// TwinCAT 3 PLC project LWLine
// Title: LINE_LJ
// Company: Aircom Automotive
// ProjectVersion: 1.0
// ProgramVersion: 3.1.4020.4
// CompilerDefines: VISU_USEWSTRING
// libraries:
//   AirLib_Mach, * (AirCom)
//   AirLib_PIM, * (AirCom)
//   VisuElemBase, * (System)
//   VisuElemMeter, * (System)
//   VisuElems, * (System)
//   VisuElemsSpecialControls, * (System)
//   VisuElemsWinControls, * (System)
//   VisuElemTextEditor, * (System)
//   VisuInputs, * (System)
//   VisuNativeControl, * (System)
//   Tc2_Math, * (Beckhoff Automation GmbH)
//   Tc2_MC2, * (Beckhoff Automation GmbH)
//   Tc2_MC2_Drive, * (Beckhoff Automation GmbH)
//   Tc2_ModbusSrv, * (Beckhoff Automation GmbH)
//   Tc2_SerialCom, * (Beckhoff Automation GmbH)
//   Tc2_TcpIp, * (Beckhoff Automation GmbH)
//   Tc3_Database, * (Beckhoff Automation GmbH)
//   TC3_EL6910_Backup_Restore, * (Beckhoff Automation GmbH)
//   Tc3_EventLogger, * (Beckhoff Automation GmbH)
//   Tc3_Interfaces, * (Beckhoff Automation GmbH)
//   Tc3_Module, * (Beckhoff Automation GmbH)
//   Util, * (System)
//   VisuDialogs, * (System)
//   VisuElemEventTable, * (System)
//   VisuGlobalClientManager, * (System)
//   VisuSymbols, * (System)
//   Tc2_EtherCAT,3.5.1.0,Beckhoff Automation GmbH
//   Tc2_Standard,newest,Beckhoff Automation GmbH
//   Tc2_System,newest,Beckhoff Automation GmbH
//   Tc2_Utilities,newest,Beckhoff Automation GmbH
//   Visu Interfaces,newest,System
//   VisuSymbols,newest,System
// project tree:
//   DUTs/DUTs/ enProductTypes_1.TcTLEO
//   DUTs/DUTs/FillingLine/ stBA02PL_Line.TcDUT
//   DUTs/DUTs/HP/ stBH0GPL_Line.TcDUT, stBH0HPL_Line.TcDUT, stBH0IPL_Line.TcDUT, stBH0JPL_Line.TcDUT, stBH0KPL_Line.TcDUT, stBH0LPL_Line.TcDUT, stBH0MPL_Line.TcDUT
//   DUTs/DUTs/PreAssembly/ stBO02PL_Line.TcDUT, stBS02PL_Line.TcDUT, stBB02PL_Line.TcDUT
//   DUTs/ enProductTypes.TcTLEO
//   / FastTask.TcTTO, GlobalTextList.TcGTLO, PIM_Task.TcTTO, PlcTask.TcTTO, Visualization Manager.TcVMO (not stored), VISU_TASK.TcTTO
//   GVLs/ Global_Alarms.TcGVL, GVL.TcGVL, GVL_Checks.TcGVL, GVL_IO.TcGVL
//   POUs/ BackgroundRS232.TcPOU, MAIN.TcPOU, SafetyBackupRestore.TcPOU
//   POUs/Checks/ CheckBounds.TcPOU, CheckDivDInt.TcPOU, CheckDivLInt.TcPOU, CheckDivLReal.TcPOU, CheckDivReal.TcPOU, CheckLRangeSigned.TcPOU, CheckLRangeUnsigned.TcPOU, CheckPointer.TcPOU, CheckRangeSigned.TcPOU, CheckRangeUnsigned.TcPOU
//   POUs/Program_PIM_Lines/ B02PL_LineBackground.TcPOU
//   POUs/Program_PIM_Lines/Filling/ BA02PL_LineBackground.TcPOU
//   POUs/Program_PIM_Lines/HP/ BH0GPL_LineBackground.TcPOU, BH0HPL_LineBackground.TcPOU, BH0IPL_LineBackground.TcPOU, BH0JPL_LineBackground.TcPOU, BH0KPL_LineBackground.TcPOU, BH0LPL_LineBackground.TcPOU, BH0MPL_LineBackground.TcPOU
//   POUs/Program_PIM_Lines/PreAssembly/ BO02PL_LineBackground.TcPOU, BS02PL_LineBackground.TcPOU, BB02PL_LineBackground.TcPOU
//   VISUs/New Visus/ HomeVisuBA02PL.TcVIS, HomeVisuBB02PL.TcVIS, HomeVisuBH0GPL.TcVIS, HomeVisuBH0HPL.TcVIS, HomeVisuBH0IPL.TcVIS, HomeVisuBH0JPL.TcVIS, HomeVisuBH0KPL.TcVIS, HomeVisuBH0LPL.TcVIS, HomeVisuBH0MPL.TcVIS, HomeVisuBO02PL.TcVIS, HomeVisuBS02PL.TcVIS, HomeVisu_1.TcVIS, vHotPlateSettings_V3_B02PL.TcVIS, vWeighingTunelVisionFrame.TcVIS
//   VISUs/ tlNames.TcTLO, tlNamesShort.TcTLO, tlStations.TcTLO
// real-time tasks:
//   TASK FastTask: cycle T#1ms, priority 20, ADS port 350
//   TASK PlcTask: cycle T#10ms, priority 22, ADS port 351
//   TASK VISU_TASK: cycle T#200000us, priority 30, ADS port 353
//   TASK PIM_Task: cycle T#10ms, priority 21, ADS port 352
// motion (NC):
//   TASK NC-Task 1 SAF: cycle T#2ms, priority 2, ADS port 501
//   TASK NC-Task 1 SVB: cycle T#10ms, priority 8, ADS port 511
//   AXIS Axis_G1_M1_Up (id 1)
//     Dynamic: Acceleration=409.623, Deceleration=409.623, Jerk=1228.87
//     Velo: RefSearch=2.73082, RefSync=2.73082, SlowManual=13.6541, FastManual=81.9246, Fast=273.082, Maximum=273.082
//     OtherSettings: AllowMotionCmdToSlave=true
//     encoder EncType=19
//       EncPara: ScaleFactorNumerator=5, ScaleFactorDenominator=1048576, MaxCount=#xffffffff
//         SoftEndMinControl: Enable=true
//         SoftEndMaxControl: Enable=true, Range=230
//         Inc: RefSearchInverse=true, RefSyncInverse=false
//     drive DrvType=16
//       DrvPara: MaxCount=#xffffffff, DriveControlDWord=#x00000100
//         Analog: VeloReferenz=300.3902, VeloScale=32, TorqueSetpointScale=10, ScaleFactorActTorque=0.1
//         TimeComp: TaskDelayCycles=1
//     controller CtrType=1
//       CtrPara: PriorControlFactor=1
//         PosDiffControl: Time=0.05
//         Observer: BandWidth=20
//   AXIS Axis_G1_M1_Dn (id 2)
//     Dynamic: Acceleration=409.623, Deceleration=409.623, Jerk=1228.87
//     Velo: RefSearch=2.73082, RefSync=2.73082, SlowManual=13.6541, FastManual=81.9246, Fast=273.082, Maximum=273.082
//     OtherSettings: AllowMotionCmdToSlave=true
//     encoder EncType=19
//       EncPara: ScaleFactorNumerator=5, ScaleFactorDenominator=1048576, MaxCount=#xffffffff
//         SoftEndMinControl: Enable=true
//         SoftEndMaxControl: Enable=true, Range=230
//         Inc: RefSearchInverse=true, RefSyncInverse=false
//     drive DrvType=16
//       DrvPara: MaxCount=#xffffffff, DriveControlDWord=#x00000100
//         Analog: VeloReferenz=300.3902, VeloScale=32, TorqueSetpointScale=10, ScaleFactorActTorque=0.1
//         TimeComp: TaskDelayCycles=1
//     controller CtrType=1
//       CtrPara: PriorControlFactor=1
//         PosDiffControl: Time=0.05
//         Observer: BandWidth=20
//   AXIS Axis_G1_M2_Up (id 3)
//     Dynamic: Acceleration=409.623, Deceleration=409.623, Jerk=1228.87
//     Velo: RefSearch=2.73082, RefSync=2.73082, SlowManual=13.6541, FastManual=81.9246, Fast=273.082, Maximum=273.082
//     OtherSettings: AllowMotionCmdToSlave=true
//     encoder EncType=19
//       EncPara: ScaleFactorNumerator=5, ScaleFactorDenominator=1048576, MaxCount=#xffffffff
//         SoftEndMinControl: Enable=true
//         SoftEndMaxControl: Enable=true, Range=230
//         Inc: RefSearchInverse=true, RefSyncInverse=false
//     drive DrvType=16
//       DrvPara: MaxCount=#xffffffff, DriveControlDWord=#x00000100
//         Analog: VeloReferenz=300.3902, VeloScale=32, TorqueSetpointScale=10, ScaleFactorActTorque=0.1
//         TimeComp: TaskDelayCycles=1
//     controller CtrType=1
//       CtrPara: PriorControlFactor=1
//         PosDiffControl: Time=0.05
//         Observer: BandWidth=20
//   AXIS Axis_G1_M2_Dn (id 4)
//     Dynamic: Acceleration=409.623, Deceleration=409.623, Jerk=1228.869
//     Velo: RefSearch=2.73082, RefSync=2.73082, SlowManual=13.6541, FastManual=81.9246, Fast=273.082, Maximum=273.082
//     OtherSettings: AllowMotionCmdToSlave=true
//     encoder EncType=19
//       EncPara: ScaleFactorNumerator=5, ScaleFactorDenominator=1048576, MaxCount=#xffffffff
//         SoftEndMinControl: Enable=true
//         SoftEndMaxControl: Enable=true, Range=230
//         Inc: RefSearchInverse=true, RefSyncInverse=false
//     drive DrvType=16
//       DrvPara: MaxCount=#xffffffff, DriveControlDWord=#x00000100
//         Analog: VeloReferenz=300.3902, VeloScale=32, TorqueSetpointScale=10, ScaleFactorActTorque=0.1
//         TimeComp: TaskDelayCycles=1
//     controller CtrType=1
//       CtrPara: PriorControlFactor=1
//         PosDiffControl: Time=0.05
//         Observer: BandWidth=20
//   AXIS Axis_G1_M3_Up (id 5)
//     Dynamic: Acceleration=409.623, Deceleration=409.623, Jerk=1228.87
//     Velo: RefSearch=2.73082, RefSync=2.73082, SlowManual=13.6541, FastManual=81.9246, Fast=273.082, Maximum=273.082
//     OtherSettings: AllowMotionCmdToSlave=true
//     encoder EncType=19
//       EncPara: ScaleFactorNumerator=5, ScaleFactorDenominator=1048576, MaxCount=#xffffffff
//         SoftEndMinControl: Enable=true
//         SoftEndMaxControl: Enable=true, Range=230
//         Inc: RefSearchInverse=true, RefSyncInverse=false
//     drive DrvType=16
//       DrvPara: MaxCount=#xffffffff, DriveControlDWord=#x00000100
//         Analog: VeloReferenz=300.3902, VeloScale=32, TorqueSetpointScale=10, ScaleFactorActTorque=0.1
//         TimeComp: TaskDelayCycles=1
//     controller CtrType=1
//       CtrPara: PriorControlFactor=1
//         PosDiffControl: Time=0.05
//         Observer: BandWidth=20
//   AXIS Axis_G1_M3_Dn (id 6)
//     Dynamic: Acceleration=409.623, Deceleration=409.623, Jerk=1228.87
//     Velo: RefSearch=2.73082, RefSync=2.73082, SlowManual=13.6541, FastManual=81.9246, Fast=273.082, Maximum=273.082
//     OtherSettings: AllowMotionCmdToSlave=true
//     encoder EncType=19
//       EncPara: ScaleFactorNumerator=5, ScaleFactorDenominator=1048576, MaxCount=#xffffffff
//         SoftEndMinControl: Enable=true
//         SoftEndMaxControl: Enable=true, Range=230
//         Inc: RefSearchInverse=true, RefSyncInverse=false
//     drive DrvType=16
//       DrvPara: MaxCount=#xffffffff, DriveControlDWord=#x00000100
//         Analog: VeloReferenz=300.3902, VeloScale=32, TorqueSetpointScale=10, ScaleFactorActTorque=0.1
//         TimeComp: TaskDelayCycles=1
//     controller CtrType=1
//       CtrPara: PriorControlFactor=1
//         PosDiffControl: Time=0.05
//         Observer: BandWidth=20
//   AXIS Axis_G2_M1_Up (id 8)
//     Dynamic: Acceleration=409.623, Deceleration=409.623, Jerk=1228.87
//     Velo: RefSearch=2.73082, RefSync=2.73082, SlowManual=13.6541, FastManual=81.9246, Fast=273.082, Maximum=273.082
//     OtherSettings: AllowMotionCmdToSlave=true
//     encoder EncType=19
//       EncPara: ScaleFactorNumerator=5, ScaleFactorDenominator=1048576, MaxCount=#xffffffff
//         SoftEndMinControl: Enable=true
//         SoftEndMaxControl: Enable=true, Range=230
//         Inc: RefSearchInverse=true, RefSyncInverse=false
//     drive DrvType=16
//       DrvPara: MaxCount=#xffffffff, DriveControlDWord=#x00000100
//         Analog: VeloReferenz=300.3902, VeloScale=32, TorqueSetpointScale=10, ScaleFactorActTorque=0.1
//         TimeComp: TaskDelayCycles=1
//     controller CtrType=1
//       CtrPara: PriorControlFactor=1
//         PosDiffControl: Time=0.15
//         Observer: BandWidth=20
//   AXIS Axis_G2_M1_Dn (id 9)
//     Dynamic: Acceleration=409.623, Deceleration=409.623, Jerk=1228.869
//     Velo: RefSearch=2.73082, RefSync=2.73082, SlowManual=13.6541, FastManual=81.9246, Fast=273.082, Maximum=273.082
//     OtherSettings: AllowMotionCmdToSlave=true
//     encoder EncType=19
//       EncPara: ScaleFactorNumerator=5, ScaleFactorDenominator=1048576, MaxCount=#xffffffff
//         SoftEndMinControl: Enable=true
//         SoftEndMaxControl: Enable=true, Range=230
//         Inc: RefSearchInverse=true, RefSyncInverse=false
//     drive DrvType=16
//       DrvPara: MaxCount=#xffffffff, DriveControlDWord=#x00000100
//         Analog: VeloReferenz=300.3902, VeloScale=32, TorqueSetpointScale=10, ScaleFactorActTorque=0.1
//         TimeComp: TaskDelayCycles=1
//     controller CtrType=1
//       CtrPara: PriorControlFactor=1
//         PosDiffControl: Time=0.15
//         Observer: BandWidth=20
//   AXIS Axis_G2_M2_Up (id 10)
//     Dynamic: Acceleration=409.623, Deceleration=409.623, Jerk=1228.87
//     Velo: RefSearch=2.73082, RefSync=2.73082, SlowManual=13.6541, FastManual=81.9246, Fast=273.082, Maximum=273.082
//     OtherSettings: AllowMotionCmdToSlave=true
//     encoder EncType=19
//       EncPara: ScaleFactorNumerator=5, ScaleFactorDenominator=1048576, MaxCount=#xffffffff
//         SoftEndMinControl: Enable=true
//         SoftEndMaxControl: Enable=true, Range=230
//         Inc: RefSearchInverse=true, RefSyncInverse=false
//     drive DrvType=16
//       DrvPara: MaxCount=#xffffffff, DriveControlDWord=#x00000100
//         Analog: VeloReferenz=300.3902, VeloScale=32, TorqueSetpointScale=10, ScaleFactorActTorque=0.1
//         TimeComp: TaskDelayCycles=1
//     controller CtrType=1
//       CtrPara: PriorControlFactor=1
//         PosDiffControl: Time=0.15
//         Observer: BandWidth=20
//   AXIS Axis_G2_M2_Dn (id 11)
//     Dynamic: Acceleration=409.623, Deceleration=409.623, Jerk=1228.869
//     Velo: RefSearch=2.73082, RefSync=2.73082, SlowManual=13.6541, FastManual=81.9246, Fast=273.082, Maximum=273.082
//     OtherSettings: AllowMotionCmdToSlave=true
//     encoder EncType=19
//       EncPara: ScaleFactorNumerator=5, ScaleFactorDenominator=1048576, MaxCount=#xffffffff
//         SoftEndMinControl: Enable=true
//         SoftEndMaxControl: Enable=true, Range=230
//         Inc: RefSearchInverse=true, RefSyncInverse=false
//     drive DrvType=16
//       DrvPara: MaxCount=#xffffffff, DriveControlDWord=#x00000100
//         Analog: VeloReferenz=300.3902, VeloScale=32, TorqueSetpointScale=10, ScaleFactorActTorque=0.1
//         TimeComp: TaskDelayCycles=1
//     controller CtrType=1
//       CtrPara: PriorControlFactor=1
//         PosDiffControl: Time=0.15
//         Observer: BandWidth=20
//   AXIS Axis_G2_M3_Up (id 12)
//     Dynamic: Acceleration=409.623, Deceleration=409.623, Jerk=1228.869
//     Velo: RefSearch=2.73082, RefSync=2.73082, SlowManual=13.6541, FastManual=81.9246, Fast=273.082, Maximum=273.082
//     OtherSettings: AllowMotionCmdToSlave=true
//     encoder EncType=19
//       EncPara: ScaleFactorNumerator=5, ScaleFactorDenominator=1048576, MaxCount=#xffffffff
//         SoftEndMinControl: Enable=true
//         SoftEndMaxControl: Enable=true, Range=230
//         Inc: RefSearchInverse=true, RefSyncInverse=false
//     drive DrvType=16
//       DrvPara: MaxCount=#xffffffff, DriveControlDWord=#x00000100
//         Analog: VeloReferenz=300.3902, VeloScale=32, TorqueSetpointScale=10, ScaleFactorActTorque=0.1
//         TimeComp: TaskDelayCycles=1
//     controller CtrType=1
//       CtrPara: PriorControlFactor=1
//         PosDiffControl: Time=0.15
//         Observer: BandWidth=20
//   AXIS Axis_G2_M3_Dn (id 13)
//     Dynamic: Acceleration=409.623, Deceleration=409.623, Jerk=1228.869
//     Velo: RefSearch=2.73082, RefSync=2.73082, SlowManual=13.6541, FastManual=81.9246, Fast=273.082, Maximum=273.082
//     OtherSettings: AllowMotionCmdToSlave=true
//     encoder EncType=19
//       EncPara: ScaleFactorNumerator=5, ScaleFactorDenominator=1048576, MaxCount=#xffffffff
//         SoftEndMinControl: Enable=true
//         SoftEndMaxControl: Enable=true, Range=230
//         Inc: RefSearchInverse=true, RefSyncInverse=false
//     drive DrvType=16
//       DrvPara: MaxCount=#xffffffff, DriveControlDWord=#x00000100
//         Analog: VeloReferenz=300.3902, VeloScale=32, TorqueSetpointScale=10, ScaleFactorActTorque=0.1
//         TimeComp: TaskDelayCycles=1
//     controller CtrType=1
//       CtrPara: PriorControlFactor=1
//         PosDiffControl: Time=0.15
//         Observer: BandWidth=20
//   AXIS Axis_G3_M1_Up (id 14)
//     Dynamic: Acceleration=409.623, Deceleration=409.623, Jerk=1228.869
//     Velo: RefSearch=2.73082, RefSync=2.73082, SlowManual=13.6541, FastManual=81.9246, Fast=273.082, Maximum=273.082
//     OtherSettings: AllowMotionCmdToSlave=true
//     encoder EncType=19
//       EncPara: ScaleFactorNumerator=5, ScaleFactorDenominator=1048576, MaxCount=#xffffffff
//         SoftEndMinControl: Enable=true
//         SoftEndMaxControl: Enable=true, Range=230
//         Inc: RefSearchInverse=true, RefSyncInverse=false
//     drive DrvType=16
//       DrvPara: MaxCount=#xffffffff, DriveControlDWord=#x00000100
//         Analog: VeloReferenz=300.3902, VeloScale=32, TorqueSetpointScale=10, ScaleFactorActTorque=0.1
//         TimeComp: TaskDelayCycles=1
//     controller CtrType=1
//       CtrPara: PriorControlFactor=1
//         PosDiffControl: Time=0.15
//         Observer: BandWidth=20
//   AXIS Axis_G3_M1_Dn (id 15)
//     Dynamic: Acceleration=409.623, Deceleration=409.623, Jerk=1228.869
//     Velo: RefSearch=2.73082, RefSync=2.73082, SlowManual=13.6541, FastManual=81.9246, Fast=273.082, Maximum=273.082
//     OtherSettings: AllowMotionCmdToSlave=true
//     encoder EncType=19
//       EncPara: ScaleFactorNumerator=5, ScaleFactorDenominator=1048576, MaxCount=#xffffffff
//         SoftEndMinControl: Enable=true
//         SoftEndMaxControl: Enable=true, Range=230
//         Inc: RefSearchInverse=true, RefSyncInverse=false
//     drive DrvType=16
//       DrvPara: MaxCount=#xffffffff, DriveControlDWord=#x00000100
//         Analog: VeloReferenz=300.3902, VeloScale=32, TorqueSetpointScale=10, ScaleFactorActTorque=0.1
//         TimeComp: TaskDelayCycles=1
//     controller CtrType=1
//       CtrPara: PriorControlFactor=1
//         PosDiffControl: Time=0.05
//         Observer: BandWidth=20
//   AXIS Axis_G3_M2_Up (id 16)
//     Dynamic: Acceleration=409.623, Deceleration=409.623, Jerk=1228.869
//     Velo: RefSearch=2.73082, RefSync=2.73082, SlowManual=13.6541, FastManual=81.9246, Fast=273.082, Maximum=273.082
//     OtherSettings: AllowMotionCmdToSlave=true
//     encoder EncType=19
//       EncPara: ScaleFactorNumerator=5, ScaleFactorDenominator=1048576, MaxCount=#xffffffff
//         SoftEndMinControl: Enable=true
//         SoftEndMaxControl: Enable=true, Range=230
//         Inc: RefSearchInverse=true, RefSyncInverse=false
//     drive DrvType=16
//       DrvPara: MaxCount=#xffffffff, DriveControlDWord=#x00000100
//         Analog: VeloReferenz=300.3902, VeloScale=32, TorqueSetpointScale=10, ScaleFactorActTorque=0.1
//         TimeComp: TaskDelayCycles=1
//     controller CtrType=1
//       CtrPara: PriorControlFactor=1
//         PosDiffControl: Time=0.05
//         Observer: BandWidth=20
//   AXIS Axis_G3_M2_Dn (id 17)
//     Dynamic: Acceleration=409.623, Deceleration=409.623, Jerk=1228.869
//     Velo: RefSearch=2.73082, RefSync=2.73082, SlowManual=13.6541, FastManual=81.9246, Fast=273.082, Maximum=273.082
//     OtherSettings: AllowMotionCmdToSlave=true
//     encoder EncType=19
//       EncPara: ScaleFactorNumerator=5, ScaleFactorDenominator=1048576, MaxCount=#xffffffff
//         SoftEndMinControl: Enable=true
//         SoftEndMaxControl: Enable=true, Range=230
//         Inc: RefSearchInverse=true, RefSyncInverse=false
//     drive DrvType=16
//       DrvPara: MaxCount=#xffffffff, DriveControlDWord=#x00000100
//         Analog: VeloReferenz=300.3902, VeloScale=32, TorqueSetpointScale=10, ScaleFactorActTorque=0.1
//         TimeComp: TaskDelayCycles=1
//     controller CtrType=1
//       CtrPara: PriorControlFactor=1
//         PosDiffControl: Time=0.05
//         Observer: BandWidth=20
//   AXIS Axis_G3_M3_Up (id 18)
//     Dynamic: Acceleration=409.623, Deceleration=409.623, Jerk=1228.87
//     Velo: RefSearch=2.73082, RefSync=2.73082, SlowManual=13.6541, FastManual=81.9246, Fast=273.082, Maximum=273.082
//     OtherSettings: AllowMotionCmdToSlave=true
//     encoder EncType=19
//       EncPara: ScaleFactorNumerator=5, ScaleFactorDenominator=1048576, MaxCount=#xffffffff
//         SoftEndMinControl: Enable=true
//         SoftEndMaxControl: Enable=true, Range=230
//         Inc: RefSearchInverse=true, RefSyncInverse=false
//     drive DrvType=16
//       DrvPara: MaxCount=#xffffffff, DriveControlDWord=#x00000100
//         Analog: VeloReferenz=300.3902, VeloScale=32, TorqueSetpointScale=10, ScaleFactorActTorque=0.1
//         TimeComp: TaskDelayCycles=1
//     controller CtrType=1
//       CtrPara: PriorControlFactor=1
//         PosDiffControl: Time=0.15
//         Observer: BandWidth=20
//   AXIS Axis_G3_M3_Dn (id 19)
//     Dynamic: Acceleration=409.623, Deceleration=409.623, Jerk=1228.869
//     Velo: RefSearch=2.73082, RefSync=2.73082, SlowManual=13.6541, FastManual=81.9246, Fast=273.082, Maximum=273.082
//     OtherSettings: AllowMotionCmdToSlave=true
//     encoder EncType=19
//       EncPara: ScaleFactorNumerator=5, ScaleFactorDenominator=1048576, MaxCount=#xffffffff
//         SoftEndMinControl: Enable=true
//         SoftEndMaxControl: Enable=true, Range=230
//         Inc: RefSearchInverse=true, RefSyncInverse=false
//     drive DrvType=16
//       DrvPara: MaxCount=#xffffffff, DriveControlDWord=#x00000100
//         Analog: VeloReferenz=300.3902, TorqueSetpointScale=10, ScaleFactorActTorque=0.1
//         TimeComp: TaskDelayCycles=1
//     controller CtrType=1
//       CtrPara: PriorControlFactor=1
//         PosDiffControl: Time=0.05
//         Observer: BandWidth=20
//   AXIS Axis_G4_M1_Up (id 7)
//     Dynamic: Acceleration=671.149, Deceleration=671.149, Jerk=2013.45
//     Velo: RefSearch=4.47433, RefSync=4.47433, SlowManual=1, FastManual=6, Fast=447.433, Maximum=447.433
//     OtherSettings: AllowMotionCmdToSlave=true
//     encoder EncType=19
//       EncPara: ScaleFactorNumerator=5, ScaleFactorDenominator=1048576, MaxCount=#xffffffff
//         SoftEndMinControl: Enable=true
//         SoftEndMaxControl: Enable=true, Range=230
//         Inc: RefSearchInverse=true, RefSyncInverse=false
//     drive DrvType=16
//       DrvPara: MaxCount=#xffffffff, DriveControlDWord=#x00000100
//         Analog: VeloReferenz=492.1763, VeloScale=32, TorqueSetpointScale=10, ScaleFactorActTorque=0.1
//         TimeComp: TaskDelayCycles=1
//     controller CtrType=1
//       CtrPara: PriorControlFactor=1
//         PosDiffControl: Time=0.05
//         Observer: BandWidth=20
//   AXIS Axis_G4_M1_Dn (id 20)
//     Dynamic: Acceleration=409.623, Deceleration=409.623, Jerk=1228.87
//     Velo: RefSearch=2.73082, RefSync=2.73082, SlowManual=13.6541, FastManual=81.9246, Fast=273.082, Maximum=273.082
//     OtherSettings: AllowMotionCmdToSlave=true
//     encoder EncType=19
//       EncPara: ScaleFactorNumerator=5, ScaleFactorDenominator=1048576, MaxCount=#xffffffff
//         SoftEndMinControl: Enable=true
//         SoftEndMaxControl: Enable=true, Range=230
//         Inc: RefSearchInverse=true, RefSyncInverse=false
//     drive DrvType=16
//       DrvPara: MaxCount=#xffffffff, DriveControlDWord=#x00000100
//         Analog: VeloReferenz=300.3902, VeloScale=32, TorqueSetpointScale=10, ScaleFactorActTorque=0.1
//         TimeComp: TaskDelayCycles=1
//     controller CtrType=1
//       CtrPara: PriorControlFactor=1
//         PosDiffControl: Time=0.05
//         Observer: BandWidth=20
//   AXIS Axis_G4_M2_Up (id 21)
//     Dynamic: Acceleration=409.623, Deceleration=409.623, Jerk=1228.87
//     Velo: RefSearch=2.73082, RefSync=2.73082, SlowManual=13.6541, FastManual=81.9246, Fast=273.082, Maximum=273.082
//     OtherSettings: AllowMotionCmdToSlave=true
//     encoder EncType=19
//       EncPara: ScaleFactorNumerator=5, ScaleFactorDenominator=1048576, MaxCount=#xffffffff
//         SoftEndMinControl: Enable=true
//         SoftEndMaxControl: Enable=true, Range=230
//         Inc: RefSearchInverse=true, RefSyncInverse=false
//     drive DrvType=16
//       DrvPara: MaxCount=#xffffffff, DriveControlDWord=#x00000100
//         Analog: VeloReferenz=300.3902, TorqueSetpointScale=10, ScaleFactorActTorque=0.1
//         TimeComp: TaskDelayCycles=1
//     controller CtrType=1
//       CtrPara: PriorControlFactor=1
//         PosDiffControl: Range=6, Time=0.15
//         Observer: BandWidth=20
//   AXIS Axis_G4_M2_Dn (id 22)
//     Dynamic: Acceleration=409.623, Deceleration=409.623, Jerk=1228.87
//     Velo: RefSearch=2.73082, RefSync=2.73082, SlowManual=13.6541, FastManual=81.9246, Fast=273.082, Maximum=273.082
//     OtherSettings: AllowMotionCmdToSlave=true
//     encoder EncType=19
//       EncPara: ScaleFactorNumerator=5, ScaleFactorDenominator=1048576, MaxCount=#xffffffff
//         SoftEndMinControl: Enable=true
//         SoftEndMaxControl: Enable=true, Range=230
//         Inc: RefSearchInverse=true, RefSyncInverse=false
//     drive DrvType=16
//       DrvPara: MaxCount=#xffffffff, DriveControlDWord=#x00000100
//         Analog: VeloReferenz=300.3902, VeloScale=32, TorqueSetpointScale=10, ScaleFactorActTorque=0.1
//         TimeComp: TaskDelayCycles=1
//     controller CtrType=1
//       CtrPara: PriorControlFactor=1
//         PosDiffControl: Range=7.5, Time=0.15
//         Observer: BandWidth=20
//   AXIS Axis_G4_M3_Up (id 23)
//     Dynamic: Acceleration=671.1495, Deceleration=671.1495, Jerk=2013.4485
//     Velo: RefSearch=4.47433, RefSync=4.47433, SlowManual=22.37165, FastManual=134.2299, Fast=447.433, Maximum=447.433
//     OtherSettings: AllowMotionCmdToSlave=true
//     encoder EncType=19
//       EncPara: ScaleFactorNumerator=5, ScaleFactorDenominator=1048576, MaxCount=#xffffffff
//         SoftEndMinControl: Enable=true
//         SoftEndMaxControl: Enable=true, Range=230
//         Inc: RefSearchInverse=true, RefSyncInverse=false
//     drive DrvType=16
//       DrvPara: MaxCount=#xffffffff, DriveControlDWord=#x00000100
//         Analog: VeloReferenz=492.1763, VeloScale=32, TorqueSetpointScale=10, ScaleFactorActTorque=0.1
//         TimeComp: TaskDelayCycles=1
//     controller CtrType=1
//       CtrPara: PriorControlFactor=1
//         PosDiffControl: Range=6, Time=0.15
//         Observer: BandWidth=20
//   AXIS Axis_G4_M3_Dn (id 24)
//     Dynamic: Acceleration=671.1495, Deceleration=671.1495, Jerk=2013.4485
//     Velo: RefSearch=4.47433, RefSync=4.47433, SlowManual=22.37165, FastManual=134.2299, Fast=447.433, Maximum=447.433
//     OtherSettings: AllowMotionCmdToSlave=true
//     encoder EncType=19
//       EncPara: ScaleFactorNumerator=5, ScaleFactorDenominator=1048576, MaxCount=#xffffffff
//         SoftEndMinControl: Enable=true
//         SoftEndMaxControl: Enable=true, Range=230
//         Inc: RefSearchInverse=true, RefSyncInverse=false
//     drive DrvType=16
//       DrvPara: MaxCount=#xffffffff, DriveControlDWord=#x00000100
//         Analog: VeloReferenz=492.1763, VeloScale=32, TorqueSetpointScale=10, ScaleFactorActTorque=0.1
//         TimeComp: TaskDelayCycles=1
//     controller CtrType=1
//       CtrPara: PriorControlFactor=1
//         PosDiffControl: Range=7.5, Time=0.15
//         Observer: BandWidth=20
//   AXIS Axis_G5_M1_Up (id 25)
//     Dynamic: Acceleration=671.149, Deceleration=671.149, Jerk=2013.45
//     Velo: RefSearch=4.47433, RefSync=4.47433, SlowManual=22.37165, FastManual=134.2299, Fast=447.433, Maximum=447.433
//     OtherSettings: AllowMotionCmdToSlave=true
//     encoder EncType=19
//       EncPara: ScaleFactorNumerator=5, ScaleFactorDenominator=1048576, MaxCount=#xffffffff
//     drive DrvType=16
//       DrvPara: MaxCount=#xffffffff, DriveControlDWord=#x00000100
//         Analog: VeloReferenz=492.1763, VeloScale=32, TorqueSetpointScale=10, ScaleFactorActTorque=0.1
//         TimeComp: TaskDelayCycles=1
//     controller CtrType=1
//       CtrPara: PriorControlFactor=1
//         Observer: BandWidth=20
//   AXIS Axis_G5_M1_Dn (id 26)
//     Dynamic: Acceleration=671.1495, Deceleration=671.1495, Jerk=2013.4485
//     Velo: RefSearch=4.47433, RefSync=4.47433, SlowManual=22.37165, FastManual=134.2299, Fast=447.433, Maximum=447.433
//     OtherSettings: AllowMotionCmdToSlave=true
//     encoder EncType=19
//       EncPara: ScaleFactorNumerator=5, ScaleFactorDenominator=1048576, MaxCount=#xffffffff
//     drive DrvType=16
//       DrvPara: MaxCount=#xffffffff, DriveControlDWord=#x00000100
//         Analog: VeloReferenz=492.1763, VeloScale=32, TorqueSetpointScale=10, ScaleFactorActTorque=0.1
//         TimeComp: TaskDelayCycles=1
//     controller CtrType=1
//       CtrPara: PriorControlFactor=1
//         Observer: BandWidth=20
//   AXIS Axis_G5_M2_Up (id 27)
//     Dynamic: Acceleration=671.1495, Deceleration=671.1495, Jerk=2013.4485
//     Velo: RefSearch=4.47433, RefSync=4.47433, SlowManual=22.37165, FastManual=134.2299, Fast=447.433, Maximum=447.433
//     OtherSettings: AllowMotionCmdToSlave=true
//     encoder EncType=19
//       EncPara: ScaleFactorNumerator=5, ScaleFactorDenominator=1048576, MaxCount=#xffffffff
//     drive DrvType=16
//       DrvPara: MaxCount=#xffffffff, DriveControlDWord=#x00000100
//         Analog: VeloReferenz=492.1763, VeloScale=32, TorqueSetpointScale=10, ScaleFactorActTorque=0.1
//         TimeComp: TaskDelayCycles=1
//     controller CtrType=1
//       CtrPara: PriorControlFactor=1
//         Observer: BandWidth=20
//   AXIS Axis_G5_M2_Dn (id 28)
//     Dynamic: Acceleration=671.1495, Deceleration=671.1495, Jerk=2013.4485
//     Velo: RefSearch=4.47433, RefSync=4.47433, SlowManual=22.37165, FastManual=134.2299, Fast=447.433, Maximum=447.433
//     OtherSettings: AllowMotionCmdToSlave=true
//     encoder EncType=19
//       EncPara: ScaleFactorNumerator=5, ScaleFactorDenominator=1048576, MaxCount=#xffffffff
//     drive DrvType=16
//       DrvPara: MaxCount=#xffffffff, DriveControlDWord=#x00000100
//         Analog: VeloReferenz=492.1763, VeloScale=32, TorqueSetpointScale=10, ScaleFactorActTorque=0.1
//         TimeComp: TaskDelayCycles=1
//     controller CtrType=1
//       CtrPara: PriorControlFactor=1
//         Observer: BandWidth=20
//   AXIS Axis_G5_M3_Up (id 29)
//     Dynamic: Acceleration=671.1495, Deceleration=671.1495, Jerk=2013.4485
//     Velo: RefSearch=4.47433, RefSync=4.47433, SlowManual=22.37165, FastManual=134.2299, Fast=447.433, Maximum=447.433
//     OtherSettings: AllowMotionCmdToSlave=true
//     encoder EncType=19
//       EncPara: ScaleFactorNumerator=5, ScaleFactorDenominator=1048576, MaxCount=#xffffffff
//     drive DrvType=16
//       DrvPara: MaxCount=#xffffffff, DriveControlDWord=#x00000100
//         Analog: VeloReferenz=492.1763, VeloScale=32, TorqueSetpointScale=10, ScaleFactorActTorque=0.1
//         TimeComp: TaskDelayCycles=1
//     controller CtrType=1
//       CtrPara: PriorControlFactor=1
//         Observer: BandWidth=20
//   AXIS Axis_G5_M3_Dn (id 30)
//     Dynamic: Acceleration=671.1495, Deceleration=671.1495, Jerk=2013.4485
//     Velo: RefSearch=4.47433, RefSync=4.47433, SlowManual=22.37165, FastManual=134.2299, Fast=447.433, Maximum=447.433
//     OtherSettings: AllowMotionCmdToSlave=true
//     encoder EncType=19
//       EncPara: ScaleFactorNumerator=5, ScaleFactorDenominator=1048576, MaxCount=#xffffffff
//     drive DrvType=16
//       DrvPara: MaxCount=#xffffffff, DriveControlDWord=#x00000100
//         Analog: VeloReferenz=492.1763, VeloScale=32, TorqueSetpointScale=10, ScaleFactorActTorque=0.1
//         TimeComp: TaskDelayCycles=1
//     controller CtrType=1
//       CtrPara: PriorControlFactor=1
//         Observer: BandWidth=20
//   AXIS Axis_G6_M1_Up (id 31)
//     Dynamic: Acceleration=671.1495, Deceleration=671.1495, Jerk=2013.4485
//     Velo: RefSearch=4.47433, RefSync=4.47433, SlowManual=22.37165, FastManual=134.2299, Fast=447.433, Maximum=447.433
//     OtherSettings: AllowMotionCmdToSlave=true
//     encoder EncType=19
//       EncPara: ScaleFactorNumerator=5, ScaleFactorDenominator=1048576, MaxCount=#xffffffff
//     drive DrvType=16
//       DrvPara: MaxCount=#xffffffff, DriveControlDWord=#x00000100
//         Analog: VeloReferenz=492.1763, VeloScale=32, TorqueSetpointScale=10, ScaleFactorActTorque=0.1
//         TimeComp: TaskDelayCycles=1
//     controller CtrType=1
//       CtrPara: PriorControlFactor=1
//         Observer: BandWidth=20
//   AXIS Axis_G6_M1_Dn (id 32)
//     Dynamic: Acceleration=671.1495, Deceleration=671.1495, Jerk=2013.4485
//     Velo: RefSearch=4.47433, RefSync=4.47433, SlowManual=22.37165, FastManual=134.2299, Fast=447.433, Maximum=447.433
//     OtherSettings: AllowMotionCmdToSlave=true
//     encoder EncType=19
//       EncPara: ScaleFactorNumerator=5, ScaleFactorDenominator=1048576, MaxCount=#xffffffff
//     drive DrvType=16
//       DrvPara: MaxCount=#xffffffff, DriveControlDWord=#x00000100
//         Analog: VeloReferenz=492.1763, VeloScale=32, TorqueSetpointScale=10, ScaleFactorActTorque=0.1
//         TimeComp: TaskDelayCycles=1
//     controller CtrType=1
//       CtrPara: PriorControlFactor=1
//         Observer: BandWidth=20
//   AXIS Axis_G6_M2_Up (id 33)
//     Dynamic: Acceleration=671.1495, Deceleration=671.1495, Jerk=2013.4485
//     Velo: RefSearch=4.47433, RefSync=4.47433, SlowManual=22.37165, FastManual=134.2299, Fast=447.433, Maximum=447.433
//     OtherSettings: AllowMotionCmdToSlave=true
//     encoder EncType=19
//       EncPara: ScaleFactorNumerator=5, ScaleFactorDenominator=1048576, MaxCount=#xffffffff
//     drive DrvType=16
//       DrvPara: MaxCount=#xffffffff, DriveControlDWord=#x00000100
//         Analog: VeloReferenz=492.1763, VeloScale=32, TorqueSetpointScale=10, ScaleFactorActTorque=0.1
//         TimeComp: TaskDelayCycles=1
//     controller CtrType=1
//       CtrPara: PriorControlFactor=1
//         Observer: BandWidth=20
//   AXIS Axis_G6_M2_Dn (id 34)
//     Dynamic: Acceleration=671.1495, Deceleration=671.1495, Jerk=2013.4485
//     Velo: RefSearch=4.47433, RefSync=4.47433, SlowManual=22.37165, FastManual=134.2299, Fast=447.433, Maximum=447.433
//     OtherSettings: AllowMotionCmdToSlave=true
//     encoder EncType=19
//       EncPara: ScaleFactorNumerator=5, ScaleFactorDenominator=1048576, MaxCount=#xffffffff
//     drive DrvType=16
//       DrvPara: MaxCount=#xffffffff, DriveControlDWord=#x00000100
//         Analog: VeloReferenz=492.1763, VeloScale=32, TorqueSetpointScale=10, ScaleFactorActTorque=0.1
//         TimeComp: TaskDelayCycles=1
//     controller CtrType=1
//       CtrPara: PriorControlFactor=1
//         Observer: BandWidth=20
//   AXIS Axis_G6_M3_Up (id 35)
//     Dynamic: Acceleration=671.1495, Deceleration=671.1495, Jerk=2013.4485
//     Velo: RefSearch=4.47433, RefSync=4.47433, SlowManual=22.37165, FastManual=134.2299, Fast=447.433, Maximum=447.433
//     OtherSettings: AllowMotionCmdToSlave=true
//     encoder EncType=19
//       EncPara: ScaleFactorNumerator=5, ScaleFactorDenominator=1048576, MaxCount=#xffffffff
//     drive DrvType=16
//       DrvPara: MaxCount=#xffffffff, DriveControlDWord=#x00000100
//         Analog: VeloReferenz=492.1763, VeloScale=32, TorqueSetpointScale=10, ScaleFactorActTorque=0.1
//         TimeComp: TaskDelayCycles=1
//     controller CtrType=1
//       CtrPara: PriorControlFactor=1
//         Observer: BandWidth=20
//   AXIS Axis_G6_M3_Dn (id 36)
//     Dynamic: Acceleration=671.1495, Deceleration=671.1495, Jerk=2013.4485
//     Velo: RefSearch=4.47433, RefSync=4.47433, SlowManual=22.37165, FastManual=134.2299, Fast=447.433, Maximum=447.433
//     OtherSettings: AllowMotionCmdToSlave=true
//     encoder EncType=19
//       EncPara: ScaleFactorNumerator=5, ScaleFactorDenominator=1048576, MaxCount=#xffffffff
//     drive DrvType=16
//       DrvPara: MaxCount=#xffffffff, DriveControlDWord=#x00000100
//         Analog: VeloReferenz=492.1763, VeloScale=32, TorqueSetpointScale=10, ScaleFactorActTorque=0.1
//         TimeComp: TaskDelayCycles=1
//     controller CtrType=1
//       CtrPara: PriorControlFactor=1
//         Observer: BandWidth=20
//   AXIS Axis_G7_M1_Up (id 37)
//     Dynamic: Acceleration=671.1495, Deceleration=671.1495, Jerk=2013.4485
//     Velo: RefSearch=4.47433, RefSync=4.47433, SlowManual=22.37165, FastManual=134.2299, Fast=447.433, Maximum=447.433
//     OtherSettings: AllowMotionCmdToSlave=true
//     encoder EncType=19
//       EncPara: ScaleFactorNumerator=5, ScaleFactorDenominator=1048576, MaxCount=#xffffffff
//     drive DrvType=16
//       DrvPara: MaxCount=#xffffffff, DriveControlDWord=#x00000100
//         Analog: VeloReferenz=492.1763, VeloScale=32, TorqueSetpointScale=10, ScaleFactorActTorque=0.1
//         TimeComp: TaskDelayCycles=1
//     controller CtrType=1
//       CtrPara: PriorControlFactor=1
//         Observer: BandWidth=20
//   AXIS Axis_G7_M1_Dn (id 38)
//     Dynamic: Acceleration=671.1495, Deceleration=671.1495, Jerk=2013.4485
//     Velo: RefSearch=4.47433, RefSync=4.47433, SlowManual=22.37165, FastManual=134.2299, Fast=447.433, Maximum=447.433
//     OtherSettings: AllowMotionCmdToSlave=true
//     encoder EncType=19
//       EncPara: ScaleFactorNumerator=5, ScaleFactorDenominator=1048576, MaxCount=#xffffffff
//     drive DrvType=16
//       DrvPara: MaxCount=#xffffffff, DriveControlDWord=#x00000100
//         Analog: VeloReferenz=492.1763, VeloScale=32, TorqueSetpointScale=10, ScaleFactorActTorque=0.1
//         TimeComp: TaskDelayCycles=1
//     controller CtrType=1
//       CtrPara: PriorControlFactor=1
//         Observer: BandWidth=20
//   AXIS Axis_G7_M2_Up (id 39)
//     Dynamic: Acceleration=102.273, Deceleration=102.273, Jerk=306.819
//     Velo: RefSearch=0.68182, RefSync=0.68182, SlowManual=3.4091, FastManual=20.4546, Fast=68.182, Maximum=447.433
//     OtherSettings: AllowMotionCmdToSlave=true
//     encoder EncType=19
//       EncPara: ScaleFactorNumerator=5, ScaleFactorDenominator=1048576, MaxCount=#xffffffff
//     drive DrvType=16
//       DrvPara: MaxCount=#xffffffff, DriveControlDWord=#x00000100
//         Analog: VeloReferenz=492.1763, TorqueSetpointScale=10, ScaleFactorActTorque=0.1
//         TimeComp: TaskDelayCycles=1
//     controller CtrType=1
//       CtrPara: PriorControlFactor=1
//         Observer: BandWidth=20
//   AXIS Axis_G7_M2_Dn (id 40)
//     Dynamic: Acceleration=102.273, Deceleration=102.273, Jerk=306.819
//     Velo: RefSearch=0.68182, RefSync=0.68182, SlowManual=3.4091, FastManual=20.4546, Fast=68.182, Maximum=447.433
//     OtherSettings: AllowMotionCmdToSlave=true
//     encoder EncType=19
//       EncPara: ScaleFactorNumerator=5, ScaleFactorDenominator=1048576, MaxCount=#xffffffff
//     drive DrvType=16
//       DrvPara: MaxCount=#xffffffff, DriveControlDWord=#x00000100
//         Analog: VeloReferenz=492.1763, TorqueSetpointScale=10, ScaleFactorActTorque=0.1
//         TimeComp: TaskDelayCycles=1
//     controller CtrType=1
//       CtrPara: PriorControlFactor=1
//         Observer: BandWidth=20
//   AXIS Axis_G7_M3_Up (id 41)
//     Dynamic: Acceleration=671.1495, Deceleration=671.1495, Jerk=2013.4485
//     Velo: RefSearch=4.47433, RefSync=4.47433, SlowManual=22.37165, FastManual=134.2299, Fast=447.433, Maximum=447.433
//     OtherSettings: AllowMotionCmdToSlave=true
//     encoder EncType=19
//       EncPara: ScaleFactorNumerator=5, ScaleFactorDenominator=1048576, MaxCount=#xffffffff
//     drive DrvType=16
//       DrvPara: MaxCount=#xffffffff, DriveControlDWord=#x00000100
//         Analog: VeloReferenz=492.1763, VeloScale=32, TorqueSetpointScale=10, ScaleFactorActTorque=0.1
//         TimeComp: TaskDelayCycles=1
//     controller CtrType=1
//       CtrPara: PriorControlFactor=1
//         Observer: BandWidth=20
//   AXIS Axis_G7_M3_Dn (id 42)
//     Dynamic: Acceleration=671.1495, Deceleration=671.1495, Jerk=2013.4485
//     Velo: RefSearch=4.47433, RefSync=4.47433, SlowManual=22.37165, FastManual=134.2299, Fast=447.433, Maximum=447.433
//     OtherSettings: AllowMotionCmdToSlave=true
//     encoder EncType=19
//       EncPara: ScaleFactorNumerator=5, ScaleFactorDenominator=1048576, MaxCount=#xffffffff
//     drive DrvType=16
//       DrvPara: MaxCount=#xffffffff, DriveControlDWord=#x00000100
//         Analog: VeloReferenz=492.1763, VeloScale=32, TorqueSetpointScale=10, ScaleFactorActTorque=0.1
//         TimeComp: TaskDelayCycles=1
//     controller CtrType=1
//       CtrPara: PriorControlFactor=1
//         Observer: BandWidth=20
//   AXIS Axis_S05_UnderPress (id 43)
//     General: UnitName=°
//     Dynamic: Acceleration=699.879, Deceleration=699.879, Jerk=2099.64
//     Velo: RefSearch=4.66586, RefSync=4.66586, SlowManual=23.3293, FastManual=139.9758, Fast=466.586, Maximum=466.586
//     OtherSettings: AllowMotionCmdToSlave=true
//     encoder EncType=19
//       EncPara: ScaleFactorNumerator=360, ScaleFactorDenominator=71303168, MaxCount=#xffffffff
//     drive DrvType=16
//       DrvPara: MaxCount=#xffffffff, DriveControlDWord=#x00000100
//         Analog: VeloReferenz=513.2446, VeloScale=32, TorqueSetpointScale=10, ScaleFactorActTorque=0.1
//         TimeComp: TaskDelayCycles=1
//     controller CtrType=1
//       CtrPara: PriorControlFactor=1
//         PosDiffControl: Range=50, Time=0.2
//         Observer: BandWidth=20
//   AXIS Rotation (id 44)
//     General: UnitName=°, UnitFlags=#x00000004
//     Dynamic: Acceleration=483.228, Deceleration=483.228, Jerk=1449.684
//     Velo: RefSearch=3.22152, RefSync=3.22152, SlowManual=16.1076, FastManual=96.6456, Fast=322.152, Maximum=322.152
//     OtherSettings: AllowMotionCmdToSlave=true
//     encoder EncType=19
//       EncPara: ScaleFactorNumerator=360, ScaleFactorDenominator=104857600, Inverse=true, MaxCount=#xffffffff
//     drive DrvType=16
//       DrvPara: Inverse=true, MaxCount=#xffffffff, DriveControlDWord=#x00020100
//         Analog: VeloReferenz=354.3672, VeloScale=32, TorqueSetpointScale=10, ScaleFactorActTorque=0.1
//         TimeComp: TaskDelayCycles=1
//     controller CtrType=1
//       CtrPara: PriorControlFactor=1
//         PosDiffControl: Range=180
//         Observer: BandWidth=20
// I/O:
//   DEVICE LAN1 (EtherCAT), AmsNetId 192.168.13.31.3.1
//     S07_RIO1 (EK1914) [EK1914, 2 Ch. Safety Input/Output 24V,  TwinSAFE]
//       modules: Module 1 (FSOE), Module 2 (DIO)
//       S07_SDI01 (EL1918) [EL1918, 8Ch. Safety Input 24V, TwinSAFE]
//         modules: Module 1 (FSOE), Module 2 (FSLOGIC)
//       S07_DI01 (EL1008) [EL1008 8Ch. Dig. Input 24V, 3ms]
//       S07_DI02 (EL1809) [EL1809 16Ch. Dig. Input 24V, 3ms]
//       S07_PWR (EL9410) [EL9410 E-Bus Power Supplier  (Diagnostics)]
//       S07_DO01 (EL2809) [EL2809 16Ch. Dig. Output 24V, 0.5A]
//       S07_LED01 (EL2564) [EL2564 4Ch. LED output, 5...48 V DC, 4 A, RGBW]
//       S07_AIO01 (EL4374) [EL4374 2Ch. Ana. Input, 2Ch. Ana. Output, +/-10V, +/-20mA, 16 Bit]
//       S07_MC1 (ELM7222-9016) [ELM7222-9016 2Ch. Servo Terminal (48 V, 8 A RMS, OCT, STO, TwinSAFE Logic)]
//         modules: Module 1 (SAFETY)
//         startup 33041:21 := 0E01 // DRV Motor Settings Ch.2 / Commutation offset
//         startup 33041:27 := 10270000 // DRV Motor Settings Ch.2 / Motor speed limitation
//         startup 33042:19 := 0000 // DRV Brake Settings Ch.2 / Emergency application timeout
//         startup 33040:51 := 0A00 // DRV Amplifier Settings Ch.2 / Stand still window
//         startup 28944:3 := 08 // DRV Outputs Ch.2 / Modes of operation
//         startup 28944:16 := FF7F // DRV Outputs Ch.2 / Positive torque limit value
//         startup 28944:17 := FF7F // DRV Outputs Ch.2 / Negative torque limit value
//         startup 33040:87 := 64 // DRV Amplifier Settings Ch.2 / Position loop velocity feed forward gain
//         startup 33040:109 := 64000000 // DRV Amplifier Settings Ch.2 / Torque feed forward gain
//         startup 28944:11 := D007 // DRV Outputs Ch.2 / Torque limitation
//         startup 33040:19 := 7600 // DRV Amplifier Settings Ch.2 / Current loop proportional gain
//         startup 33040:18 := 1300 // DRV Amplifier Settings Ch.2 / Current loop integral time
//         startup 33040:21 := 23010000 // DRV Amplifier Settings Ch.2 / Velocity loop proportional gain
//         startup 33040:20 := 96000000 // DRV Amplifier Settings Ch.2 / Velocity loop integral time
//       S07_T1 (ELM3502-0000) [ELM3502-0000 2Ch. Bridge Measuring (SG), 24 bit, high precision]
//       S07_ETH1 (EL6614) [EL6614 4 Port Switch (Ethernet, CoE)]
//       Term 401 (EL9011) [EL9011 End Terminal]
//   DEVICE Device 1 (ECAT EIP Scanner (EL6652)), AmsNetId 192.168.13.31.2.1
//     Box 2 (SS5 Series) // <INFO> </INFO> <EDS> C:\TwinCAT\3.1\Config\Io\EtherNetIP\Irayple_SS5_1.2.eds </EDS>
// variable links:
//   LWLine/LWLine Instance <-> Device 1 (ECAT EIP Scanner (EL6652))/Box 2 (SS5 Series)
//     PlcTask Inputs/MAIN.fbSmartCamera.arInputData @bit {8..1600 step 8} <-> Connection 1 (Input/Output)/Inputs/Input Data_{5..204}  (200 links)
//     PlcTask Inputs/MAIN.fbSmartCamera.arInputData <-> Connection 1 (Input/Output)/Inputs/Input Data_4
//     PlcTask Inputs/MAIN.fbSmartCamera.arTotalRunning <-> Connection 1 (Input/Output)/Inputs/Input Data
//     PlcTask Inputs/MAIN.fbSmartCamera.arTotalRunning @bit 8 <-> Connection 1 (Input/Output)/Inputs/Input Data_1
//     PlcTask Inputs/MAIN.fbSmartCamera.arTotalRunning @bit 16 <-> Connection 1 (Input/Output)/Inputs/Input Data_2
//     PlcTask Inputs/MAIN.fbSmartCamera.arTotalRunning @bit 24 <-> Connection 1 (Input/Output)/Inputs/Input Data_3
//     PlcTask Outputs/MAIN.fbSmartCamera.usiResetStatistic <-> Connection 1 (Input/Output)/Outputs/Ouput Data_1
//     PlcTask Outputs/MAIN.fbSmartCamera.usiSwitchProjectID <-> Connection 1 (Input/Output)/Outputs/Ouput Data_2
//     PlcTask Outputs/MAIN.fbSmartCamera.usiTrigger <-> Connection 1 (Input/Output)/Outputs/Ouput Data
//   LWLine/LWLine Instance <-> LAN1 (EtherCAT)
//     PIM_Task Inputs/MAIN.stLine_BA02PL.fbLine.fbEtherCAT_Diag.sSystemNetIDLink <-> InfoData/AmsNetId
//     PIM_Task Inputs/MAIN.stLine_BB02PL.fbLine.fbEtherCAT_Diag.sSystemNetIDLink <-> InfoData/AmsNetId
//     PIM_Task Inputs/MAIN.stLine_BH0GPL.fbLine.fbEtherCAT_Diag.sSystemNetIDLink <-> InfoData/AmsNetId
//     PIM_Task Inputs/MAIN.stLine_BH0IPL.fbLine.fbEtherCAT_Diag.sSystemNetIDLink <-> InfoData/AmsNetId
//     PIM_Task Inputs/MAIN.stLine_BH0JPL.fbLine.fbEtherCAT_Diag.sSystemNetIDLink <-> InfoData/AmsNetId
//     PIM_Task Inputs/MAIN.stLine_BH0KPL.fbLine.fbEtherCAT_Diag.sSystemNetIDLink <-> InfoData/AmsNetId
//     PIM_Task Inputs/MAIN.stLine_BH0LPL.fbLine.fbEtherCAT_Diag.sSystemNetIDLink <-> InfoData/AmsNetId
//     PIM_Task Inputs/MAIN.stLine_BH0MPL.fbLine.fbEtherCAT_Diag.sSystemNetIDLink <-> InfoData/AmsNetId
//     PIM_Task Inputs/MAIN.stLine_BO02PL.fbLine.fbEtherCAT_Diag.sSystemNetIDLink <-> InfoData/AmsNetId
//     PIM_Task Inputs/MAIN.stLine_BS02PL.fbLine.fbEtherCAT_Diag.sSystemNetIDLink <-> InfoData/AmsNetId
//     PlcTask Inputs/MAIN.stLine_BH0HPL.fbLine.fbEtherCAT_Diag.sSystemNetIDLink <-> InfoData/AmsNetId
//   LWLine/LWLine Instance <-> LAN1 (EtherCAT)/S07_RIO1 (EK1914)
//     PIM_Task Inputs/MAIN.stLine_BA02PL.stStation_BA02PL07.fbStation.fbElectricyCounter.bElectricyUsageCounter <-> Module 2 (DIO)/DIO Inputs/Input 0
//     PlcTask Inputs/MAIN.fbWeighingTunel.stInOuts.bI_SafetyReset_1 <-> Module 2 (DIO)/DIO Inputs/Input 1
//     PlcTask Inputs/MAIN.fbWeighingTunel.stInOuts.bI_SafetyReset_2 <-> Module 2 (DIO)/DIO Inputs/Input 2
//   LWLine/LWLine Instance <-> LAN1 (EtherCAT)/S07_RIO1 (EK1914)/S07_AIO01 (EL4374)
//     PlcTask Inputs/MAIN.fbWeighingTunel.fbLoadingStation.stInOuts.iBottleDetectionSensor <-> AI Standard (INT16) Channel 1/Value
//     PlcTask Outputs/MAIN.fbWeighingTunel.fbUnloadingStation.fbConveyor.iQ_ConveyorSpeedOut <-> AO Standard (INT16) Channel 3/Value
//   LWLine/LWLine Instance <-> LAN1 (EtherCAT)/S07_RIO1 (EK1914)/S07_DI01 (EL1008)
//     PlcTask Inputs/MAIN.fbWeighingTunel.fbTableAxis.bHomingSensor <-> Channel 4/Input
//     PlcTask Inputs/MAIN.fbWeighingTunel.fbUnloadingStation.fbConveyor.bI_ConveyorOnFeedback <-> Channel 5/Input
//     PlcTask Inputs/MAIN.fbWeighingTunel.fbUnloadingStation.fbUnloadingSensor.bI_SensorSignal <-> Channel 3/Input
//     PlcTask Inputs/MAIN.fbWeighingTunel.fbWeighingStation.fbBottleDrawerSensor.bI_SensorSignal <-> Channel 2/Input
//     PlcTask Inputs/MAIN.fbWeighingTunel.fbWeighingStation.fbBottleSensor.bI_SensorSignal <-> Channel 1/Input
//   LWLine/LWLine Instance <-> LAN1 (EtherCAT)/S07_RIO1 (EK1914)/S07_DI02 (EL1809)
//     PlcTask Inputs/MAIN.fbWeighingTunel.fbLoadingStation.fbSeparator1.bI_HomePosition <-> Channel 7/Input
//     PlcTask Inputs/MAIN.fbWeighingTunel.fbLoadingStation.fbSeparator2.bI_HomePosition <-> Channel 8/Input
//     PlcTask Inputs/MAIN.fbWeighingTunel.fbLoadingStation.fbSeparator1_Sensor.bI_SensorSignal <-> Channel 9/Input
//     PlcTask Inputs/MAIN.fbWeighingTunel.fbLoadingStation.fbSeparator2_Sensor.bI_SensorSignal <-> Channel 10/Input
//     PlcTask Inputs/MAIN.fbWeighingTunel.fbUnloadingStation.fbUnloadingActuator.bI_HomePosition <-> Channel 3/Input
//     PlcTask Inputs/MAIN.fbWeighingTunel.fbUnloadingStation.fbUnloadingActuator.bI_WorkPosition <-> Channel 4/Input
//     PlcTask Inputs/MAIN.fbWeighingTunel.fbWeighingStation.fbPusherActuator.bI_HomePosition <-> Channel 1/Input
//     PlcTask Inputs/MAIN.fbWeighingTunel.fbWeighingStation.fbPusherActuator.bI_WorkPosition <-> Channel 2/Input
//     PlcTask Inputs/MAIN.fbWeighingTunel.fbWeighingStation.fbWeighingActuator.bI_HomePosition <-> Channel 6/Input
//     PlcTask Inputs/MAIN.fbWeighingTunel.fbWeighingStation.fbWeighingActuator.bI_WorkPosition <-> Channel 5/Input
//   LWLine/LWLine Instance <-> LAN1 (EtherCAT)/S07_RIO1 (EK1914)/S07_DO01 (EL2809)
//     PlcTask Outputs/MAIN.fbWeighingTunel.fbLoadingStation.fbSeparator1.bQ_Work <-> Channel 13/Output
//     PlcTask Outputs/MAIN.fbWeighingTunel.fbLoadingStation.fbSeparator2.bQ_Work <-> Channel 12/Output
//     PlcTask Outputs/MAIN.fbWeighingTunel.fbUnloadingStation.fbConveyor.bQ_ConveyorON <-> Channel 9/Output
//     PlcTask Outputs/MAIN.fbWeighingTunel.fbUnloadingStation.fbUnloadingActuator.bQ_Work <-> Channel 8/Output
//     PlcTask Outputs/MAIN.fbWeighingTunel.fbWeighingStation.fbPusherActuator.bQ_Work <-> Channel 6/Output
//     PlcTask Outputs/MAIN.fbWeighingTunel.fbWeighingStation.fbWeighingActuator.bQ_Work <-> Channel 7/Output
//     PlcTask Outputs/MAIN.fbWeighingTunel.stInOuts.bQ_LampBlue <-> Channel 3/Output
//     PlcTask Outputs/MAIN.fbWeighingTunel.stInOuts.bQ_LampGreen <-> Channel 5/Output
//     PlcTask Outputs/MAIN.fbWeighingTunel.stInOuts.bQ_LampRed <-> Channel 2/Output
//     PlcTask Outputs/MAIN.fbWeighingTunel.stInOuts.bQ_LampWhite <-> Channel 1/Output
//     PlcTask Outputs/MAIN.fbWeighingTunel.stInOuts.bQ_LampYellow <-> Channel 4/Output
//     PlcTask Outputs/MAIN.fbWeighingTunel.stInOuts.bQ_ResetLamp_1 <-> Channel 10/Output
//     PlcTask Outputs/MAIN.fbWeighingTunel.stInOuts.bQ_ResetLamp_2 <-> Channel 11/Output
//   LWLine/LWLine Instance <-> LAN1 (EtherCAT)/S07_RIO1 (EK1914)/S07_MC1 (ELM7222-9016)
//     PlcTask Outputs/MAIN.fbWeighingTunel.fbTableAxis.bQ_ToSafety_ErrorAck <-> Module 1 (SAFETY)/SAFETY Standard Outputdata/Standard In Var 3
//     PlcTask Outputs/MAIN.fbWeighingTunel.fbTableAxis.bQ_ToSafety_Run <-> Module 1 (SAFETY)/SAFETY Standard Outputdata/Standard In Var 2
//   LWLine/LWLine Instance <-> LAN1 (EtherCAT)/S07_RIO1 (EK1914)/S07_T1 (ELM3502-0000)
//     FastTask Inputs/MAIN.fbWeighingTunel.fbWeighingStation.fbWeighing.arrSamples[1] <-> PAI Samples 1 Channel 1/Samples[0]
//   LWLine/LWLine Instance <-> NC-Task 1 SAF/Axes/Axis_G1_M1_Dn
//     PlcTask Inputs/MAIN.fbHotPlate_G1_M1.fbAxisDn.stInOuts.stAxis_Data.NcToPlc <-> Outputs/ToPlc
//     PlcTask Outputs/MAIN.fbHotPlate_G1_M1.fbAxisDn.stInOuts.stAxis_Data.PlcToNc <-> Inputs/FromPlc
//   LWLine/LWLine Instance <-> NC-Task 1 SAF/Axes/Axis_G1_M1_Up
//     PlcTask Inputs/MAIN.fbHotPlate_G1_M1.fbAxisUp.stInOuts.stAxis_Data.NcToPlc <-> Outputs/ToPlc
//     PlcTask Outputs/MAIN.fbHotPlate_G1_M1.fbAxisUp.stInOuts.stAxis_Data.PlcToNc <-> Inputs/FromPlc
//   LWLine/LWLine Instance <-> NC-Task 1 SAF/Axes/Axis_G1_M2_Dn
//     PlcTask Inputs/MAIN.fbHotPlate_G1_M2.fbAxisDn.stInOuts.stAxis_Data.NcToPlc <-> Outputs/ToPlc
//     PlcTask Outputs/MAIN.fbHotPlate_G1_M2.fbAxisDn.stInOuts.stAxis_Data.PlcToNc <-> Inputs/FromPlc
//   LWLine/LWLine Instance <-> NC-Task 1 SAF/Axes/Axis_G1_M2_Up
//     PlcTask Inputs/MAIN.fbHotPlate_G1_M2.fbAxisUp.stInOuts.stAxis_Data.NcToPlc <-> Outputs/ToPlc
//     PlcTask Outputs/MAIN.fbHotPlate_G1_M2.fbAxisUp.stInOuts.stAxis_Data.PlcToNc <-> Inputs/FromPlc
//   LWLine/LWLine Instance <-> NC-Task 1 SAF/Axes/Axis_G1_M3_Dn
//     PlcTask Inputs/MAIN.fbHotPlate_G1_M3.fbAxisDn.stInOuts.stAxis_Data.NcToPlc <-> Outputs/ToPlc
//     PlcTask Outputs/MAIN.fbHotPlate_G1_M3.fbAxisDn.stInOuts.stAxis_Data.PlcToNc <-> Inputs/FromPlc
//   LWLine/LWLine Instance <-> NC-Task 1 SAF/Axes/Axis_G1_M3_Up
//     PlcTask Inputs/MAIN.fbHotPlate_G1_M3.fbAxisUp.stInOuts.stAxis_Data.NcToPlc <-> Outputs/ToPlc
//     PlcTask Outputs/MAIN.fbHotPlate_G1_M3.fbAxisUp.stInOuts.stAxis_Data.PlcToNc <-> Inputs/FromPlc
//   LWLine/LWLine Instance <-> NC-Task 1 SAF/Axes/Axis_G2_M1_Dn
//     PlcTask Inputs/MAIN.fbHotPlate_G2_M1.fbAxisDn.stInOuts.stAxis_Data.NcToPlc <-> Outputs/ToPlc
//     PlcTask Outputs/MAIN.fbHotPlate_G2_M1.fbAxisDn.stInOuts.stAxis_Data.PlcToNc <-> Inputs/FromPlc
//   LWLine/LWLine Instance <-> NC-Task 1 SAF/Axes/Axis_G2_M1_Up
//     PlcTask Inputs/MAIN.fbHotPlate_G2_M1.fbAxisUp.stInOuts.stAxis_Data.NcToPlc <-> Outputs/ToPlc
//     PlcTask Outputs/MAIN.fbHotPlate_G2_M1.fbAxisUp.stInOuts.stAxis_Data.PlcToNc <-> Inputs/FromPlc
//   LWLine/LWLine Instance <-> NC-Task 1 SAF/Axes/Axis_G2_M2_Dn
//     PlcTask Inputs/MAIN.fbHotPlate_G2_M2.fbAxisDn.stInOuts.stAxis_Data.NcToPlc <-> Outputs/ToPlc
//     PlcTask Outputs/MAIN.fbHotPlate_G2_M2.fbAxisDn.stInOuts.stAxis_Data.PlcToNc <-> Inputs/FromPlc
//   LWLine/LWLine Instance <-> NC-Task 1 SAF/Axes/Axis_G2_M2_Up
//     PlcTask Inputs/MAIN.fbHotPlate_G2_M2.fbAxisUp.stInOuts.stAxis_Data.NcToPlc <-> Outputs/ToPlc
//     PlcTask Outputs/MAIN.fbHotPlate_G2_M2.fbAxisUp.stInOuts.stAxis_Data.PlcToNc <-> Inputs/FromPlc
//   LWLine/LWLine Instance <-> NC-Task 1 SAF/Axes/Axis_G2_M3_Dn
//     PlcTask Inputs/MAIN.fbHotPlate_G2_M3.fbAxisDn.stInOuts.stAxis_Data.NcToPlc <-> Outputs/ToPlc
//     PlcTask Outputs/MAIN.fbHotPlate_G2_M3.fbAxisDn.stInOuts.stAxis_Data.PlcToNc <-> Inputs/FromPlc
//   LWLine/LWLine Instance <-> NC-Task 1 SAF/Axes/Axis_G2_M3_Up
//     PlcTask Inputs/MAIN.fbHotPlate_G2_M3.fbAxisUp.stInOuts.stAxis_Data.NcToPlc <-> Outputs/ToPlc
//     PlcTask Outputs/MAIN.fbHotPlate_G2_M3.fbAxisUp.stInOuts.stAxis_Data.PlcToNc <-> Inputs/FromPlc
//   LWLine/LWLine Instance <-> NC-Task 1 SAF/Axes/Axis_G3_M1_Dn
//     PlcTask Inputs/MAIN.fbHotPlate_G3_M1.fbAxisDn.stInOuts.stAxis_Data.NcToPlc <-> Outputs/ToPlc
//     PlcTask Outputs/MAIN.fbHotPlate_G3_M1.fbAxisDn.stInOuts.stAxis_Data.PlcToNc <-> Inputs/FromPlc
//   LWLine/LWLine Instance <-> NC-Task 1 SAF/Axes/Axis_G3_M1_Up
//     PlcTask Inputs/MAIN.fbHotPlate_G3_M1.fbAxisUp.stInOuts.stAxis_Data.NcToPlc <-> Outputs/ToPlc
//     PlcTask Outputs/MAIN.fbHotPlate_G3_M1.fbAxisUp.stInOuts.stAxis_Data.PlcToNc <-> Inputs/FromPlc
//   LWLine/LWLine Instance <-> NC-Task 1 SAF/Axes/Axis_G3_M2_Dn
//     PlcTask Inputs/MAIN.fbHotPlate_G3_M2.fbAxisDn.stInOuts.stAxis_Data.NcToPlc <-> Outputs/ToPlc
//     PlcTask Outputs/MAIN.fbHotPlate_G3_M2.fbAxisDn.stInOuts.stAxis_Data.PlcToNc <-> Inputs/FromPlc
//   LWLine/LWLine Instance <-> NC-Task 1 SAF/Axes/Axis_G3_M2_Up
//     PlcTask Inputs/MAIN.fbHotPlate_G3_M2.fbAxisUp.stInOuts.stAxis_Data.NcToPlc <-> Outputs/ToPlc
//     PlcTask Outputs/MAIN.fbHotPlate_G3_M2.fbAxisUp.stInOuts.stAxis_Data.PlcToNc <-> Inputs/FromPlc
//   LWLine/LWLine Instance <-> NC-Task 1 SAF/Axes/Axis_G3_M3_Dn
//     PlcTask Inputs/MAIN.fbHotPlate_G3_M3.fbAxisDn.stInOuts.stAxis_Data.NcToPlc <-> Outputs/ToPlc
//     PlcTask Outputs/MAIN.fbHotPlate_G3_M3.fbAxisDn.stInOuts.stAxis_Data.PlcToNc <-> Inputs/FromPlc
//   LWLine/LWLine Instance <-> NC-Task 1 SAF/Axes/Axis_G3_M3_Up
//     PlcTask Inputs/MAIN.fbHotPlate_G3_M3.fbAxisUp.stInOuts.stAxis_Data.NcToPlc <-> Outputs/ToPlc
//     PlcTask Outputs/MAIN.fbHotPlate_G3_M3.fbAxisUp.stInOuts.stAxis_Data.PlcToNc <-> Inputs/FromPlc
//   LWLine/LWLine Instance <-> NC-Task 1 SAF/Axes/Axis_G4_M1_Dn
//     PlcTask Inputs/MAIN.fbHotPlate_G4_M1.fbAxisDn.stInOuts.stAxis_Data.NcToPlc <-> Outputs/ToPlc
//     PlcTask Outputs/MAIN.fbHotPlate_G4_M1.fbAxisDn.stInOuts.stAxis_Data.PlcToNc <-> Inputs/FromPlc
//   LWLine/LWLine Instance <-> NC-Task 1 SAF/Axes/Axis_G4_M1_Up
//     PlcTask Inputs/MAIN.fbHotPlate_G4_M1.fbAxisUp.stInOuts.stAxis_Data.NcToPlc <-> Outputs/ToPlc
//     PlcTask Outputs/MAIN.fbHotPlate_G4_M1.fbAxisUp.stInOuts.stAxis_Data.PlcToNc <-> Inputs/FromPlc
//   LWLine/LWLine Instance <-> NC-Task 1 SAF/Axes/Axis_G4_M2_Dn
//     PlcTask Inputs/MAIN.fbHotPlate_G4_M2.fbAxisDn.stInOuts.stAxis_Data.NcToPlc <-> Outputs/ToPlc
//     PlcTask Outputs/MAIN.fbHotPlate_G4_M2.fbAxisDn.stInOuts.stAxis_Data.PlcToNc <-> Inputs/FromPlc
//   LWLine/LWLine Instance <-> NC-Task 1 SAF/Axes/Axis_G4_M2_Up
//     PlcTask Inputs/MAIN.fbHotPlate_G4_M2.fbAxisUp.stInOuts.stAxis_Data.NcToPlc <-> Outputs/ToPlc
//     PlcTask Outputs/MAIN.fbHotPlate_G4_M2.fbAxisUp.stInOuts.stAxis_Data.PlcToNc <-> Inputs/FromPlc
//   LWLine/LWLine Instance <-> NC-Task 1 SAF/Axes/Axis_G4_M3_Dn
//     PlcTask Inputs/MAIN.fbHotPlate_G4_M3.fbAxisDn.stInOuts.stAxis_Data.NcToPlc <-> Outputs/ToPlc
//     PlcTask Outputs/MAIN.fbHotPlate_G4_M3.fbAxisDn.stInOuts.stAxis_Data.PlcToNc <-> Inputs/FromPlc
//   LWLine/LWLine Instance <-> NC-Task 1 SAF/Axes/Axis_G4_M3_Up
//     PlcTask Inputs/MAIN.fbHotPlate_G4_M3.fbAxisUp.stInOuts.stAxis_Data.NcToPlc <-> Outputs/ToPlc
//     PlcTask Outputs/MAIN.fbHotPlate_G4_M3.fbAxisUp.stInOuts.stAxis_Data.PlcToNc <-> Inputs/FromPlc
//   LWLine/LWLine Instance <-> NC-Task 1 SAF/Axes/Axis_G5_M1_Dn
//     PlcTask Inputs/MAIN.fbHotPlate_G5_M1.fbAxisDn.stInOuts.stAxis_Data.NcToPlc <-> Outputs/ToPlc
//     PlcTask Outputs/MAIN.fbHotPlate_G5_M1.fbAxisDn.stInOuts.stAxis_Data.PlcToNc <-> Inputs/FromPlc
//   LWLine/LWLine Instance <-> NC-Task 1 SAF/Axes/Axis_G5_M1_Up
//     PlcTask Inputs/MAIN.fbHotPlate_G5_M1.fbAxisUp.stInOuts.stAxis_Data.NcToPlc <-> Outputs/ToPlc
//     PlcTask Outputs/MAIN.fbHotPlate_G5_M1.fbAxisUp.stInOuts.stAxis_Data.PlcToNc <-> Inputs/FromPlc
//   LWLine/LWLine Instance <-> NC-Task 1 SAF/Axes/Axis_G5_M2_Dn
//     PlcTask Inputs/MAIN.fbHotPlate_G5_M2.fbAxisDn.stInOuts.stAxis_Data.NcToPlc <-> Outputs/ToPlc
//     PlcTask Outputs/MAIN.fbHotPlate_G5_M2.fbAxisDn.stInOuts.stAxis_Data.PlcToNc <-> Inputs/FromPlc
//   LWLine/LWLine Instance <-> NC-Task 1 SAF/Axes/Axis_G5_M2_Up
//     PlcTask Inputs/MAIN.fbHotPlate_G5_M2.fbAxisUp.stInOuts.stAxis_Data.NcToPlc <-> Outputs/ToPlc
//     PlcTask Outputs/MAIN.fbHotPlate_G5_M2.fbAxisUp.stInOuts.stAxis_Data.PlcToNc <-> Inputs/FromPlc
//   LWLine/LWLine Instance <-> NC-Task 1 SAF/Axes/Axis_G5_M3_Dn
//     PlcTask Inputs/MAIN.fbHotPlate_G5_M3.fbAxisDn.stInOuts.stAxis_Data.NcToPlc <-> Outputs/ToPlc
//     PlcTask Outputs/MAIN.fbHotPlate_G5_M3.fbAxisDn.stInOuts.stAxis_Data.PlcToNc <-> Inputs/FromPlc
//   LWLine/LWLine Instance <-> NC-Task 1 SAF/Axes/Axis_G5_M3_Up
//     PlcTask Inputs/MAIN.fbHotPlate_G5_M3.fbAxisUp.stInOuts.stAxis_Data.NcToPlc <-> Outputs/ToPlc
//     PlcTask Outputs/MAIN.fbHotPlate_G5_M3.fbAxisUp.stInOuts.stAxis_Data.PlcToNc <-> Inputs/FromPlc
//   LWLine/LWLine Instance <-> NC-Task 1 SAF/Axes/Axis_G6_M1_Dn
//     PlcTask Inputs/MAIN.fbHotPlate_G6_M1.fbAxisDn.stInOuts.stAxis_Data.NcToPlc <-> Outputs/ToPlc
//     PlcTask Outputs/MAIN.fbHotPlate_G6_M1.fbAxisDn.stInOuts.stAxis_Data.PlcToNc <-> Inputs/FromPlc
//   LWLine/LWLine Instance <-> NC-Task 1 SAF/Axes/Axis_G6_M1_Up
//     PlcTask Inputs/MAIN.fbHotPlate_G6_M1.fbAxisUp.stInOuts.stAxis_Data.NcToPlc <-> Outputs/ToPlc
//     PlcTask Outputs/MAIN.fbHotPlate_G6_M1.fbAxisUp.stInOuts.stAxis_Data.PlcToNc <-> Inputs/FromPlc
//   LWLine/LWLine Instance <-> NC-Task 1 SAF/Axes/Axis_G6_M2_Dn
//     PlcTask Inputs/MAIN.fbHotPlate_G6_M2.fbAxisDn.stInOuts.stAxis_Data.NcToPlc <-> Outputs/ToPlc
//     PlcTask Outputs/MAIN.fbHotPlate_G6_M2.fbAxisDn.stInOuts.stAxis_Data.PlcToNc <-> Inputs/FromPlc
//   LWLine/LWLine Instance <-> NC-Task 1 SAF/Axes/Axis_G6_M2_Up
//     PlcTask Inputs/MAIN.fbHotPlate_G6_M2.fbAxisUp.stInOuts.stAxis_Data.NcToPlc <-> Outputs/ToPlc
//     PlcTask Outputs/MAIN.fbHotPlate_G6_M2.fbAxisUp.stInOuts.stAxis_Data.PlcToNc <-> Inputs/FromPlc
//   LWLine/LWLine Instance <-> NC-Task 1 SAF/Axes/Axis_G6_M3_Dn
//     PlcTask Inputs/MAIN.fbHotPlate_G6_M3.fbAxisDn.stInOuts.stAxis_Data.NcToPlc <-> Outputs/ToPlc
//     PlcTask Outputs/MAIN.fbHotPlate_G6_M3.fbAxisDn.stInOuts.stAxis_Data.PlcToNc <-> Inputs/FromPlc
//   LWLine/LWLine Instance <-> NC-Task 1 SAF/Axes/Axis_G6_M3_Up
//     PlcTask Inputs/MAIN.fbHotPlate_G6_M3.fbAxisUp.stInOuts.stAxis_Data.NcToPlc <-> Outputs/ToPlc
//     PlcTask Outputs/MAIN.fbHotPlate_G6_M3.fbAxisUp.stInOuts.stAxis_Data.PlcToNc <-> Inputs/FromPlc
//   LWLine/LWLine Instance <-> NC-Task 1 SAF/Axes/Axis_G7_M1_Dn
//     PlcTask Inputs/MAIN.fbHotPlate_G7_M1.fbAxisDn.stInOuts.stAxis_Data.NcToPlc <-> Outputs/ToPlc
//     PlcTask Outputs/MAIN.fbHotPlate_G7_M1.fbAxisDn.stInOuts.stAxis_Data.PlcToNc <-> Inputs/FromPlc
//   LWLine/LWLine Instance <-> NC-Task 1 SAF/Axes/Axis_G7_M1_Up
//     PlcTask Inputs/MAIN.fbHotPlate_G7_M1.fbAxisUp.stInOuts.stAxis_Data.NcToPlc <-> Outputs/ToPlc
//     PlcTask Outputs/MAIN.fbHotPlate_G7_M1.fbAxisUp.stInOuts.stAxis_Data.PlcToNc <-> Inputs/FromPlc
//   LWLine/LWLine Instance <-> NC-Task 1 SAF/Axes/Axis_G7_M2_Dn
//     PlcTask Inputs/MAIN.fbHotPlate_G7_M2.fbAxisDn.stInOuts.stAxis_Data.NcToPlc <-> Outputs/ToPlc
//     PlcTask Outputs/MAIN.fbHotPlate_G7_M2.fbAxisDn.stInOuts.stAxis_Data.PlcToNc <-> Inputs/FromPlc
//   LWLine/LWLine Instance <-> NC-Task 1 SAF/Axes/Axis_G7_M2_Up
//     PlcTask Inputs/MAIN.fbHotPlate_G7_M2.fbAxisUp.stInOuts.stAxis_Data.NcToPlc <-> Outputs/ToPlc
//     PlcTask Outputs/MAIN.fbHotPlate_G7_M2.fbAxisUp.stInOuts.stAxis_Data.PlcToNc <-> Inputs/FromPlc
//   LWLine/LWLine Instance <-> NC-Task 1 SAF/Axes/Axis_G7_M3_Dn
//     PlcTask Inputs/MAIN.fbHotPlate_G7_M3.fbAxisDn.stInOuts.stAxis_Data.NcToPlc <-> Outputs/ToPlc
//     PlcTask Outputs/MAIN.fbHotPlate_G7_M3.fbAxisDn.stInOuts.stAxis_Data.PlcToNc <-> Inputs/FromPlc
//   LWLine/LWLine Instance <-> NC-Task 1 SAF/Axes/Axis_G7_M3_Up
//     PlcTask Inputs/MAIN.fbHotPlate_G7_M3.fbAxisUp.stInOuts.stAxis_Data.NcToPlc <-> Outputs/ToPlc
//     PlcTask Outputs/MAIN.fbHotPlate_G7_M3.fbAxisUp.stInOuts.stAxis_Data.PlcToNc <-> Inputs/FromPlc
//   LWLine/LWLine Instance <-> NC-Task 1 SAF/Axes/Axis_S05_UnderPress
//     PlcTask Inputs/MAIN.fb_UnderPressure_Tester_Machine.fbAxis.stAxisReference.NcToPlc <-> Outputs/ToPlc
//     PlcTask Outputs/MAIN.fb_UnderPressure_Tester_Machine.fbAxis.stAxisReference.PlcToNc <-> Inputs/FromPlc
//   LWLine/LWLine Instance <-> NC-Task 1 SAF/Axes/Rotation
//     PlcTask Inputs/MAIN.fbWeighingTunel.fbTableAxis.stAxis_Data.NcToPlc <-> Outputs/ToPlc
//     PlcTask Outputs/MAIN.fbWeighingTunel.fbTableAxis.stAxis_Data.PlcToNc <-> Inputs/FromPlc
//   Axes/Rotation <-> LAN1 (EtherCAT)/S07_RIO1 (EK1914)/S07_MC1 (ELM7222-9016)
//     Drive/Inputs/In/nDataIn1 <-> DRV Following error actual value Channel 2/Following error actual value
//     Drive/Inputs/In/nDcOutputTime <-> InfoData/DcOutputShift
//     Drive/Inputs/In/nState1 <-> DRV Statusword Channel 2/Statusword
//     Drive/Inputs/In/nState2 <-> DRV Statusword Channel 2/Statusword @bit 8
//     Drive/Inputs/In/nState4 @bit 1 <-> WcState/InputToggle0
//     Drive/Inputs/In/nState4 <-> WcState/WcState0
//     Drive/Outputs/Out/nCtrl1 <-> DRV Controlword Channel 2/Controlword
//     Drive/Outputs/Out/nCtrl2 <-> DRV Controlword Channel 2/Controlword @bit 8
//     Drive/Outputs/Out/nDataOut1 <-> DRV Target position Channel 2/Target position
//     Drive/Outputs/Out/nDataOut4[0] <-> DRV Target torque Channel 2/Target torque
//     Enc/Inputs/In/nDataIn1 <-> FB Position Channel 2/Position
//     Enc/Inputs/In/nDcInputTime <-> InfoData/DcInputShift
//     Enc/Inputs/In/nState4 @bit 1 <-> WcState/InputToggle0
//     Enc/Inputs/In/nState4 <-> WcState/WcState0

CONFIGURATION LWLine
    RESOURCE PLC ON TwinCAT3
        TASK FastTask(INTERVAL := T#1ms, PRIORITY := 20);
        TASK PIM_Task(INTERVAL := T#10ms, PRIORITY := 21);
        TASK PlcTask(INTERVAL := T#10ms, PRIORITY := 22);
        TASK VISU_TASK(INTERVAL := T#200000us, PRIORITY := 30);
        PROGRAM BackgroundRS232 WITH FastTask : BackgroundRS232;
        PROGRAM B02PL_LineBackground WITH PIM_Task : B02PL_LineBackground;
        PROGRAM MAIN WITH PlcTask : MAIN;
        PROGRAM VisuElems_Visu_Prg WITH VISU_TASK : VisuElems.Visu_Prg;
    END_RESOURCE
END_CONFIGURATION

// ---- DUTs/DUTs/enProductTypes_1.TcTLEO
{attribute 'qualified_only'}
{attribute 'strict'}
{attribute 'to_string'}
TYPE enProductTypes_1 :
(
	_PSA := 1,
	PORSCHE_992 := 2,
	VOLVO_SPA := 3,
	_8P0 := 4,
	JAGUAR_FGA_TC02_0040 := 0,	// -> 0
	HAOS_FGA_TC01_0006 := 5,	// -> 5
	NISSAN_FGA_TC01_0007:= 6,	// -> 6
	MERCEDES:= 7,				// -> 7
	FGA_TC02_0049 := 8,
	MAZDA := 9,
	SUBARU := 10,
	BC4 := 11
);
END_TYPE

// ---- DUTs/DUTs/FillingLine/stBA02PL_Line.TcDUT
TYPE stBA02PL_Line EXTENDS stPIM_LineEventsModule :
STRUCT
	{attribute 'OPC.UA.DA' := '1'}
	stStation_BA02PL01 : stPIM_StationEventsModule_2_Machine;
	{attribute 'OPC.UA.DA' := '1'}
	stStation_BA02PL02 : stPIM_StationEventsModule_1_Machine;
	{attribute 'OPC.UA.DA' := '1'}
	stStation_BA02PL03 : stPIM_StationEventsModule_1_Machine;
	{attribute 'OPC.UA.DA' := '1'}
	stStation_BA02PL04 : stPIM_StationEventsModule_1_Machine;
	{attribute 'OPC.UA.DA' := '1'}
	stStation_BA02PL05 : stPIM_StationEventsModule_1_Machine;
	{attribute 'OPC.UA.DA' := '1'}
	stStation_BA02PL06 : stPIM_StationEventsModule_2_Machine;
	{attribute 'OPC.UA.DA' := '1'}
	stStation_BA02PL07 : stPIM_StationEventsModule_1_Machine;
END_STRUCT
END_TYPE

// ---- DUTs/DUTs/HP/stBH0GPL_Line.TcDUT
TYPE stBH0GPL_Line EXTENDS stPIM_LineEventsModule :
STRUCT

	{attribute 'OPC.UA.DA' := '1'}
	stStation_BH0GPL01 : stPIM_StationEventsModule_3_Machine;
END_STRUCT
END_TYPE

// ---- DUTs/DUTs/HP/stBH0HPL_Line.TcDUT
TYPE stBH0HPL_Line EXTENDS stPIM_LineEventsModule :
STRUCT

	{attribute 'OPC.UA.DA' := '1'}
	stStation_BH0HPL01 : stPIM_StationEventsModule_3_Machine;
END_STRUCT
END_TYPE

// ---- DUTs/DUTs/HP/stBH0IPL_Line.TcDUT
TYPE stBH0IPL_Line EXTENDS stPIM_LineEventsModule :
STRUCT

	{attribute 'OPC.UA.DA' := '1'}
	stStation_BH0IPL01 : stPIM_StationEventsModule_3_Machine;
END_STRUCT
END_TYPE

// ---- DUTs/DUTs/HP/stBH0JPL_Line.TcDUT
TYPE stBH0JPL_Line EXTENDS stPIM_LineEventsModule :
STRUCT

	{attribute 'OPC.UA.DA' := '1'}
	stStation_BH0JPL01 : stPIM_StationEventsModule_3_Machine;
END_STRUCT
END_TYPE

// ---- DUTs/DUTs/HP/stBH0KPL_Line.TcDUT
TYPE stBH0KPL_Line EXTENDS stPIM_LineEventsModule :
STRUCT

	{attribute 'OPC.UA.DA' := '1'}
	stStation_BH0KPL01 : stPIM_StationEventsModule_3_Machine;
END_STRUCT
END_TYPE

// ---- DUTs/DUTs/HP/stBH0LPL_Line.TcDUT
TYPE stBH0LPL_Line EXTENDS stPIM_LineEventsModule :
STRUCT

	{attribute 'OPC.UA.DA' := '1'}
	stStation_BH0LPL01 : stPIM_StationEventsModule_3_Machine;
END_STRUCT
END_TYPE

// ---- DUTs/DUTs/HP/stBH0MPL_Line.TcDUT
TYPE stBH0MPL_Line EXTENDS stPIM_LineEventsModule :
STRUCT

	{attribute 'OPC.UA.DA' := '1'}
	stStation_BH0MPL01 : stPIM_StationEventsModule_3_Machine;
END_STRUCT
END_TYPE

// ---- DUTs/DUTs/PreAssembly/stBO02PL_Line.TcDUT
TYPE stBO02PL_Line EXTENDS stPIM_LineEventsModule :
STRUCT

	{attribute 'OPC.UA.DA' := '1'}
	stStation_BO02PL01 : stPIM_StationEventsModule_1_Machine;
	{attribute 'OPC.UA.DA' := '1'}
	stStation_BO02PL02 : stPIM_StationEventsModule_1_Machine;
END_STRUCT
END_TYPE

// ---- DUTs/DUTs/PreAssembly/stBS02PL_Line.TcDUT
TYPE stBS02PL_Line EXTENDS stPIM_LineEventsModule :
STRUCT

	{attribute 'OPC.UA.DA' := '1'}
	stStation_BS02PL01 : stPIM_StationEventsModule_1_Machine;
END_STRUCT
END_TYPE

// ---- DUTs/DUTs/PreAssembly/stBB02PL_Line.TcDUT
TYPE stBB02PL_Line EXTENDS stPIM_LineEventsModule :
STRUCT

	{attribute 'OPC.UA.DA' := '1'}
	stStation_BB02PL01 : stPIM_StationEventsModule_1_Machine;
END_STRUCT
END_TYPE

// ---- DUTs/enProductTypes.TcTLEO
{attribute 'qualified_only'}
{attribute 'strict'}
{attribute 'to_string'}
TYPE enProductTypes :
(
	LK3G3_4G0C := 0,
	LK3G3_4L0A := 1
);
END_TYPE

// ---- GVLs/Global_Alarms.TcGVL
VAR_GLOBAL CONSTANT
	FIRST_MESSAGE: UDINT := 1;
	LAST_MESSAGE: UDINT := 1200;
END_VAR
VAR_GLOBAL
	MSG_ALARM_List			:ARRAY[FIRST_MESSAGE..LAST_MESSAGE] OF BOOL;
	MSG_ALARM_ListQuit		:ARRAY[FIRST_MESSAGE..LAST_MESSAGE] OF BOOL;
	MSG_WARNING_List		:ARRAY[FIRST_MESSAGE..LAST_MESSAGE] OF BOOL;
	MSG_WARNING_ListQuit	:ARRAY[FIRST_MESSAGE..LAST_MESSAGE] OF BOOL;
	aAlarms					:ARRAY[1..80] OF ST_ReadEvent;
END_VAR

// ---- GVLs/GVL.TcGVL
//{attribute 'Tc2GvlVarNames'}
VAR_GLOBAL CONSTANT
	// Określenie wyglądu dla każdego rodzaju alarmu - 
	iAlarmClassesQty:INT:= 7;
	astAlarmColorTable:ARRAY [1 .. iAlarmClassesQty] OF stAlarmRowAppearanceData:= [
		(sFontName:='Arial', iFontSize:=10, dwFontFlags:=0, dwTextColor:=16#FF404040, dwAlignmentFlags:=0, dwBackgroundColor:=16#FFCDCDCD, dwFrameColor:=16#FF585858, iFrameWidth:= 1),	// Info
		(sFontName:='Arial', iFontSize:=10, dwFontFlags:=0, dwTextColor:=16#FF404040, dwAlignmentFlags:=0, dwBackgroundColor:=16#FFCDCDCD, dwFrameColor:=16#FF585858, iFrameWidth:= 1),	// Warning
		(sFontName:='Arial', iFontSize:=10, dwFontFlags:=0, dwTextColor:=16#FF404040, dwAlignmentFlags:=0, dwBackgroundColor:=16#FFCDCDCD, dwFrameColor:=16#FF585858, iFrameWidth:= 1),	// Error
		(sFontName:='Arial', iFontSize:=10, dwFontFlags:=0, dwTextColor:=16#FF404040, dwAlignmentFlags:=0, dwBackgroundColor:=16#FFCDCDCD, dwFrameColor:=16#FF585858, iFrameWidth:= 1),	// Quality
		(sFontName:='Arial', iFontSize:=10, dwFontFlags:=0, dwTextColor:=16#FF404040, dwAlignmentFlags:=0, dwBackgroundColor:=16#FFCDCDCD, dwFrameColor:=16#FF585858, iFrameWidth:= 1),	// Maintenance
		(sFontName:='Arial', iFontSize:=10, dwFontFlags:=0, dwTextColor:=16#FF404040, dwAlignmentFlags:=0, dwBackgroundColor:=16#FFCDCDCD, dwFrameColor:=16#FF585858, iFrameWidth:= 1),	// IT
		(sFontName:='Arial', iFontSize:=10, dwFontFlags:=0, dwTextColor:=16#FF404040, dwAlignmentFlags:=0, dwBackgroundColor:=16#FFCDCDCD, dwFrameColor:=16#FF585858, iFrameWidth:= 1)	// Developer
		]; 
	// https://www.rapidtables.com/convert/color/rgb-to-hex.html
END_VAR


VAR_GLOBAL PERSISTENT
	nProductType:enProductTypes;
	sCurrentLanguage:STRING(10);
	
	// S01
	stS01_PressSettings:stSonicPress_MachSettings_V4_1;
	stS01_TestParams:stSonicPress_TestParams_V4_1;
	
	// S02
	stS02_PressSettings:stSonicPress_MachSettings_V4_1;
	stS02_TestParams:stSonicPress_TestParams_V4_1;
	
	// S03
	stS03_PressSettings:stSonicPress_MachSettings_V4_1;
	stS03_TestParams:stSonicPress_TestParams_V4_1;
	
	// S04
	stS04_PressSettings:stSonicPress_MachSettings_V4_1;
	stS04_TestParams:stSonicPress_TestParams_V4_1;

	abChoseStationsToLog:ARRAY [1.. 22] OF BOOL :=[22(TRUE)]; 
	
	// Zmienne systemu wizyjnego - nie usuwać oraz nie zmieniać
	//CA
	diProductTypeCA05PL:DINT;
	sReferenceDataMatrixTextCA05PL:STRING(80);
	diReferenceStickerTypeCA05PL:DINT;
	bReferenceSignValueCA05PL:BOOL;
	//CP
	diProductTypeCP05PL:DINT;
	sReferenceDataMatrixTextCP05PL:STRING(80);
	diReferenceStickerTypeCP05PL:DINT;
	bReferenceSignValueCP05PL:BOOL;
	
	//Bottle filling line
	
	//S_01 Test
	
	//S_01                              	
	st_Filler_A_Parameters					: stModTcpSlaveParams_V3_1;
	st_Cork_Parameters						: stModTcpSlaveParams_V3_1;
	//S_02
	st_1_SonicTech_USWelderSettings			: stSonicTech_MachSettings_V4_1;
	//S_03
	st_Filler_B_Parameters					: stModTcpSlaveParams_V3_1;
	//S_04	
	st_2_SonicTech_USWelderSettings			: stSonicTech_MachSettings_V4_1;
	//S_05	
	st_UnderPressureTester_Params			: stUnderPressureTestParams_V3_1;
	stUnderPressureTestParams				: stUnderPressureTestParams_V3_1;
	stUnderPressureTestStatus				: stUnderPressureTestStatus_V3_1;
	//S_06	
	st_Sticker_Parameters					: stModTcpSlaveParams_V3_1;
	st_Laser_Parameters						: stModTcpSlaveParams_V3_2;
	//S_09	
	st_Tunel_Params							: stDetectionTunelParams_V3_1;
END_VAR
VAR_GLOBAL
	// Common Data
	bCompressedAirCtrSaveTrigger:BOOL;
	bEnergyConsCtrSaveTrigger:BOOL;
	rCompressedAirCounter:REAL;
	bLogDataTrigger:BOOL;
	fbAlarmMasterTable:fbAlarmMasterTable;		// Logowanie błędów - nie usuwać!!!
	fbStringFormat:FB_FormatString;
END_VAR

// ---- GVLs/GVL_Checks.TcGVL
{attribute 'qualified_only'}
VAR_GLOBAL PERSISTENT
	diCheckBounds			: DINT;	(*Licznik przekroczen zakresu indexow, np. tablic*)
	diCheckDivDInt			: DINT;	(*Licznik prob dzielenia Dint przez 0*)
	diCheckDivLInt			: DINT; (*Licznik prob dzielenia LInt przez 0*)
	diCheckDivLReal			: DINT; (*Licznik prob dzielenia LREAL przez 0*)
	diCheckDivReal			: DINT; (*Licznik prob dzielenia REAL przez 0*)
	diCheckLRangeSigned		: DINT;	(*Licznik przekroczen liczby znakowej duży zakres*)
	diCheckLRangeUnsigned	: DINT; (*Licznik przekroczen liczby bezznakowej duży zakres*)
	diCheckRangeSigned		: DINT;	(*Licznik przekroczen liczby znakowej*)
	diCheckRangeUnsigned	: DINT; (*Licznik przekroczen liczby bezznakowej*)
	diCheckPointer			: DINT; 
END_VAR

// ---- GVLs/GVL_IO.TcGVL
VAR_GLOBAL

//******************** Strona I ********************  
	bCompressedAirFlowImpulse AT %I* : BOOL;		// Impuls co 30L
	bCompressedAirFlowAlarmHigh AT %I* : BOOL;		// Alarm gdy przekroczony przepływ 300L/min
	bCompressedAirFlowImpulsePreAssembly			AT %I* :BOOL;
	bCompressedAirFlowImpulseFilling	 			AT %I* :BOOL;
	bCompressedAirFlowImpulseHotPlate	 			AT %I* :BOOL;
// Komunikacja RS485
// S01
	stS01_1_BearingPress_IO				: stSonicPress_DigInOuts_V4_1;
	bS01_Trigger			 			AT %Q* :BOOL;
	bS01_Result 						AT %I* :BOOL;
	bS01_Ready	 						AT %I* :BOOL;
	
// S02	- 
	stS02_1_BearingPress_IO				: stSonicPress_DigInOuts_V4_1;
	
// S03 - 
	stS03_1_BearingPress_IO				: stSonicPress_DigInOuts_V4_1;
	stS03_CapFixture_IO					: stCapDetectionInOuts;
// S04 - 
	stS04_1_BearingPress_IO				: stSonicPress_DigInOuts_V4_1;
	
	
// Sxx Plug A - 
	stSxxA_1_PlugAWelder_IO				: stSonicTech_DigInOuts_V3_1;
	
	
// Sxx Plug B - 
	stSxxB_1_PlugAWelder_IO				: stSonicTech_DigInOuts_V3_1;
//	Bottle filling line
		//S02
	b_1_SonicTech_EnergyConsumptionImp 				AT %I* :BOOL;
	st_1_SonicTech_WeldingMachine_IO				: stSonicTech_DigInOuts_V4_1;
	//S04
	b_2_SonicTech_EnergyConsumptionImp 				AT %I* :BOOL;
	st_2_SonicTech_WeldingMachine_IO				: stSonicTech_DigInOuts_V4_1;
	//S05
	stUnderPreserInOuts 							: stUnderPressureTesterInOuts_V3_1;
	stTransporterInOuts								: stTransporterInOuts_V3_2;
	stUnderPressureInOuts_V2						: stUnderPressureTesterInOuts_V3_1;
	//S07
	stTunelInOuts									: stDetectionTunelInOuts_V3_1;
	stSerialData_S02_S04 				: stSerialComData;
END_VAR

// ---- POUs/BackgroundRS232.TcPOU
PROGRAM BackgroundRS232
VAR
	
END_VAR

GVL_IO.stSerialData_S02_S04.fbSerialCom(RxBufferEL:=GVL_IO.stSerialData_S02_S04.RxBufferEL,TxBufferEL:=GVL_IO.stSerialData_S02_S04.TxBufferEL);
MAIN.fbWeighingTunel.fbWeighingStation.fbWeighing();

END_PROGRAM

// ---- POUs/MAIN.TcPOU
PROGRAM MAIN
VAR	
	{attribute 'OPC.UA.DA' := '0'}
	 
	//  stStation_L{nazwa linii}_S{nazwa stanowiska}[_M{numer maszyny}]
	//  Stanowisko S01
	{attribute 'OPC.UA.DA' := '0'}
	fbS01_BearingPress: fbSonicPress_V4_1;
	{attribute 'OPC.UA.DA' := '0'}
	fbS01_KeyencePNVisSens: fbSealingCorkAssKeyencePN_V4_1;
	// 	Stanowisko S02 
	{attribute 'OPC.UA.DA' := '0'}
	fbS02_BearingPress: fbSonicPress_V4_1;
	// 	Stanowisko S03 
	{attribute 'OPC.UA.DA' := '0'}
	fbS03_BearingPress: fbSonicPress_V4_1;
	{attribute 'OPC.UA.DA' := '0'}
	fbS03_CapFixture	: fbCapDetectionFixture_V4_1;
	// 	Stanowisko S04
	{attribute 'OPC.UA.DA' := '0'}
	fbS04_BearingPress: fbSonicPress_V4_1;
	// HotPlate G1
	{attribute 'OPC.UA.DA' := '0'}
	fbHotPlate_G1_M1: fbHP_Control_V3_1;
	{attribute 'OPC.UA.DA' := '0'}
	fbHotPlate_G1_M2: fbHP_Control_V3_1;
	{attribute 'OPC.UA.DA' := '0'}
	fbHotPlate_G1_M3: fbHP_Control_V3_1;
	// HotPlate G2
	{attribute 'OPC.UA.DA' := '0'}
	fbHotPlate_G2_M1: fbHP_Control_V3_1;
	{attribute 'OPC.UA.DA' := '0'}
	fbHotPlate_G2_M2: fbHP_Control_V3_1;
	{attribute 'OPC.UA.DA' := '0'}
	fbHotPlate_G2_M3: fbHP_Control_V3_1;
	// HotPlate G3
	{attribute 'OPC.UA.DA' := '0'}
	fbHotPlate_G3_M1: fbHP_Control_V3_1;
	{attribute 'OPC.UA.DA' := '0'}
	fbHotPlate_G3_M2: fbHP_Control_V3_1;
	{attribute 'OPC.UA.DA' := '0'}
	fbHotPlate_G3_M3: fbHP_Control_V3_1;
	// HotPlate G4
	{attribute 'OPC.UA.DA' := '0'}
	fbHotPlate_G4_M1: fbHP_Control_V3_1;
	{attribute 'OPC.UA.DA' := '0'}
	fbHotPlate_G4_M2: fbHP_Control_V3_1;
	{attribute 'OPC.UA.DA' := '0'}
	fbHotPlate_G4_M3: fbHP_Control_V3_1;
	// HotPlate G5
	{attribute 'OPC.UA.DA' := '0'}
	fbHotPlate_G5_M1: fbHP_Control_V3_1;
	{attribute 'OPC.UA.DA' := '0'}
	fbHotPlate_G5_M2: fbHP_Control_V3_1;
	{attribute 'OPC.UA.DA' := '0'}
	fbHotPlate_G5_M3: fbHP_Control_V3_1;
	// HotPlate G6
	{attribute 'OPC.UA.DA' := '0'}
	fbHotPlate_G6_M1: fbHP_Control_V3_1;
	{attribute 'OPC.UA.DA' := '0'}
	fbHotPlate_G6_M2: fbHP_Control_V3_1;
	{attribute 'OPC.UA.DA' := '0'}
	fbHotPlate_G6_M3: fbHP_Control_V3_1;
	// HotPlate G7
	{attribute 'OPC.UA.DA' := '0'}
	fbHotPlate_G7_M1: fbHP_Control_V3_1;
	{attribute 'OPC.UA.DA' := '0'}
	fbHotPlate_G7_M2: fbHP_Control_V3_1;
	{attribute 'OPC.UA.DA' := '0'}
	fbHotPlate_G7_M3: fbHP_Control_V3_1;
	// Dla całej linii
	fbS_TONAirFlowAlarm:TON;
	fbS_AirFlowAlarmTrigger:R_TRIG;
	
	fbIISReset:fbIIS_Restart;
	bRestart_IIS: BOOL;
	bRomErrorTableReset: BOOL;
	fbTcWcfReset: fbTcAdsWcfHost_Restart;
	bRestartTcWcf:BOOL;
	fbSonicModbus		: fbModbusCore;
	bResetWcfAtStartup: BOOL;
	bTrigger: BOOL;
	//fbModbusTcpCore	: fbModTCP_Core;
	//Bottle filling line
		//ACT_1_Filler_A
			//fb_Filler_A_Machine : fbChiniseMachine(I_Pim := fb_Filler_A_Station);
			{attribute 'OPC.UA.DA' := '0'}
			fb_Filler_A_Machine : fbChiniseMachine_v3_1; 
		//ACT_2_Cork
			{attribute 'OPC.UA.DA' := '0'}
			fb_Cork_Machine : fbChiniseMachine_v3_1;
		//ACT_3_SonicTech
			{attribute 'OPC.UA.DA' := '0'}
			fb_1_SonicTech_SonictechUSW		: fbSonictechUSWM_V4_1;
			fbModbusCoreS02_S04				: fbModbusCore;
		//ACT_4_Filler_B
			{attribute 'OPC.UA.DA' := '0'}
			fb_Filler_B_Machine : fbChiniseMachine_v3_1;
		//ACT_5_SonicTech
			{attribute 'OPC.UA.DA' := '0'}
			fb_2_SonicTech_SonictechUSW: fbSonictechUSWM_V4_1;
		//ACT_6_UnderPressure_Tester
			{attribute 'OPC.UA.DA' := '0'}
			fbTransporterUnderpressure	: fbTransporter_V3_2;
			{attribute 'OPC.UA.DA' := '0'}
			fb_UnderPressure_Tester_Machine : fbVacuumChamber_V3_2;
		//ACT_7_Sticker
			{attribute 'OPC.UA.DA' := '0'}
			fb_Sticker_Machine : fbChiniseMachine_v3_1;
		//ACT_8_Laser
			{attribute 'OPC.UA.DA' := '0'}
			fb_Laser_Machine : fbChiniseMachine_Laser_V3_2;
			{attribute 'OPC.UA.DA' := '0'}
			fb_Laser_TCP: FB_TCP_SendString;
			{attribute 'OPC.UA.DA' := '0'}
			fb_Laser_TCP_Manual: FB_TCP_SendStringManualTest;
	//ACT_9_Tunel
	{attribute 'OPC.UA.DA' := '0'}
	fbWeighingTunel				:FB_WeighingTunel;
	fbVision					:fbIRaypleVision;
	fbSmartCamera				:fbIRaypleSmartCamera;
	stSmartCameraParams			:stIraypleSmartCameraParams;
	{attribute 'OPC.UA.DA' := '0'}		
	fbS01_EthDiagnose				: fbTerminalDiagnoser;
	{attribute 'OPC.UA.DA' := '0'}
	fbS03_EthDiagnose				: fbTerminalDiagnoser;
	{attribute 'OPC.UA.DA' := '0'}
	fbS06_EthDiagnose				: fbTerminalDiagnoser;
	{attribute 'OPC.UA.DA' := '0'}
	fbPressS01_ProfinetDiagnose		: fbTerminalDiagnoser;
	{attribute 'OPC.UA.DA' := '0'}
	fbS03Press_EthDiagnose			: fbTerminalDiagnoser;
END_VAR
VAR
	//Filling Line
	{attribute 'OPC.UA.DA' := '1'}
	stLine_BA02PL				: stBA02PL_Line;{attribute 'OPC.UA.DA' := '1'}
	//PreAssembly
	{attribute 'OPC.UA.DA' := '1'}
	stLine_BO02PL				: stBO02PL_Line;
	{attribute 'OPC.UA.DA' := '1'}
	stLine_BS02PL				: stBS02PL_Line;
	{attribute 'OPC.UA.DA' := '1'}
	stLine_BB02PL				: stBB02PL_Line;
	//HP
	{attribute 'OPC.UA.DA' := '1'}
	stLine_BH0GPL				: stBH0GPL_Line;
	{attribute 'OPC.UA.DA' := '1'}
	stLine_BH0HPL				: stBH0HPL_Line;
	{attribute 'OPC.UA.DA' := '1'}
	stLine_BH0IPL				: stBH0IPL_Line;
	{attribute 'OPC.UA.DA' := '1'}
	stLine_BH0JPL				: stBH0JPL_Line;
	{attribute 'OPC.UA.DA' := '1'}
	stLine_BH0KPL				: stBH0KPL_Line;
	{attribute 'OPC.UA.DA' := '1'}
	stLine_BH0LPL				: stBH0LPL_Line;
	{attribute 'OPC.UA.DA' := '1'}
	stLine_BH0MPL				: stBH0MPL_Line;
END_VAR
VAR PERSISTENT
	bKeepSQLConnected: BOOL := TRUE;
	iMaxSimCmdNumber: INT := 3;
	nProductTypeMemory: enProductTypes;
END_VAR

//B02PL_LineBackground();
fbModbusCoreS02_S04(stSerialData:=GVL_IO.stSerialData_S02_S04);
// ************* Elementy wspólne dla wszystkich stanowisk	*************
PLC_BaseFunctions();
SafetyBackupRestore();
// Alarmowanie - tablica alarmów (GVL.fbErrorsHistoryTable) jest obsługiwana poprzez metody - funkcja nie musi być wywoływana
GVL.bLogDataTrigger := GVL_Aircom.stAC_DT_Data.bNew_Second_IMP;
fbSonicModbus(stSerialData:=GVL_IO.stSerialData_S02_S04);

// Restart usługi odpowiadającej za wizualizację WWW
fbIISReset(bExecute := bRestart_IIS);
bRestart_IIS R=fbIISReset.bBusy;

// Restart serwisu odpowiadającego za komunikację z PIM oraz PC-stickami systemówizyjnych
bResetWcfAtStartup S= bRestartTcWcf S= GVL_Aircom.stAC_DT_Data.diPLC_UpTimeSeconds = 30 AND NOT bResetWcfAtStartup;		// Automatyczny reset po włączeniu zasilania
fbTcWcfReset(bExecute := bRestartTcWcf);

// Czyszczenie historii alarmów
IF bRomErrorTableReset THEN
	GVL.fbAlarmMasterTable.mReset();
	bRomErrorTableReset:= FALSE;
END_IF

//Rdzeń komunikacji Modbus TCP
//fbModbusTcpCore(stTimeStruct:=GVL_Aircom.stAC_DT_Data);
// Przełączanie pomiędzy parametrami
//ACT_SelProdType();

// ************* Obsługa stanowisk - kolejny Act_LN.. to kolejne stanowisko	*************
//fbSonicTechCom_1Part(stData := GVL_IO.stRS485_Part_I, tTimeout := T#1S, uiResendQty := 1);
ACT_S01();	// Prasa SonicTech
ACT_S02();	// Prasa SonicTech
ACT_S03();	// Prasa SonicTech
ACT_S04();	// Prasa SonicTech - montaż łożysk w kole
//Filing Line
ACT_1_Filler_A();
ACT_2_Cork();
ACT_3_SonicTech();
ACT_4_Filler_B();
ACT_5_SonicTech();
ACT_6_UnderPressure_Tester();
ACT_7_Sticker();

ACT_9_WeighingTunel();

ACT_8_Laser();





ACT_HP1();
ACT_HP2();
ACT_HP3();
ACT_HP4();
ACT_HP5();
ACT_HP6();
ACT_HP7();

// Zużycie sprężonego powietrza oraz wybów częstotliwości zapisu
GVL.bCompressedAirCtrSaveTrigger := GVL_Aircom.stAC_DT_Data.bNew_Shift;
GVL.bEnergyConsCtrSaveTrigger := GVL_Aircom.stAC_DT_Data.bNew_Shift;


fbS_TONAirFlowAlarm(IN:= GVL_IO.bCompressedAirFlowAlarmHigh, PT:= T#5S);
fbS_AirFlowAlarmTrigger(CLK:= fbS_TONAirFlowAlarm.Q);
IF fbS_AirFlowAlarmTrigger.Q THEN
	GVL.fbAlarmMasterTable.mPushRow(nAlarmClass:= enAlarmClasses.Error, sMachineId := 'L_Line', sEventDesc := 'High Air Flow Alarm Active' , dwErrorId := 0);	
END_IF

sCurrentLanguage := VisuElems.CURRENTLANGUAGE;
	
//Nowe liczneie
//ACT_SideAirMeasure();
// Kontrola etherCAT
fbS01_EthDiagnose();
fbS03_EthDiagnose();
fbS06_EthDiagnose();
fbPressS01_ProfinetDiagnose();
fbS03Press_EthDiagnose();

ACTION _OpisProgramu_Notatki:
(*		
*************************************************************************************************************************************************************************************************************
ToDo:
- Auto zmiana prarametrów
- GRBL skalowanie tekstu
- Timeout zapytania sql w kolejce
- Wdrożyć podejście DRY Dont Repeat Yourself



*************************************************************************************************************************************************************************************************************
1. Opis algorytmu pracy z PIM:		


Wspólne numery kroków w algorytmach pracy 
0 - Krok inicjalizacyjny
5 - Krok spoczynkowy w którym algorytm oczekuje na nową operację

70 - Zapis statusu - ustawienie zmiennych i wystawienie bitów
71 - Oczekiwanie na zapis statusu
75 - Zapis statusu i danych rozszerzonych - ustawienie zmiennych i wystawienie bitów
76 - Oczekiwanie na zapis statusu


90 - Nowy błąd z zapisem statusu - ustawiany bit zapisu statusu 
91 - Oczekiwanie na zapis statusu - ustawiany bit bBlokowanieStanowsika

92 - Nowy błąd bez zapisu statusu (dodatkowy kod błędu) z wymaganym potwierdzeniem przez min. operatora - ustawiany bit bAlarmStanowiska
93 - Nowy błąd bez zapisu statusu - potwierdzenie przez operatora lub automatyczne przez PLC
99 - Oczekiwanie na potwierdzenie błędu przez PIM


*************************************************************************************************************************************************************************************************************
2. Zmiany w programie:

2022.03.31 - Wprowadzenie bitu bAlarmStanowiska, uaktualnienie algorytmów pracy z opcją włączenia wymagania zapisu statusu do DB




*************************************************************************************************************************************************************************************************************
Notatki:
Znaczenie poszczególnych zmiennych
 MachineSettings - Ustawienia maszyny nie związane z parametrami operacji/testów 
 MachineWorkParameters - Parametry konfiguracyjne cyklu maszyny (czas pompowania, energia zgrzewu itp)
 
 
Interfejs z systemem PIM powinien zapewniać:
- sprawdzenie czy jest zezwolenie na pracę

Teksty do wyświetlenia w kompilatorze
{text 'Tekst do wyświetlenia'}
{info 'Tekst do wyświetlenia'}
{warning 'Tekst do wyświetlenia'}
{error 'Tekst do wyświetlenia'}

*)
END_ACTION

ACTION ACT_1_Filler_A:
GVL.st_Filler_A_Parameters.bPartsCount:= TRUE;
GVL.st_Filler_A_Parameters.iErrorOffset := 1000;
GVL.st_Filler_A_Parameters.iPort:= 500;
GVL.st_Filler_A_Parameters.iUnitId := 1;
GVL.st_Filler_A_Parameters.sIpAdress := '192.168.13.180';
GVL.st_Filler_A_Parameters.iRegisterReadStartAdress:=9000;
GVL.st_Filler_A_Parameters.iRegisterWriteStartAdress:=9020;
GVL.st_Filler_A_Parameters.iRegisterReadAmount := 20;
GVL.st_Filler_A_Parameters.iRegisterWriteAmount := 20;
GVL.st_Filler_A_Parameters.sMachineIdenfier := 'BA02PL01_M1';

fb_Filler_A_Machine(
stLine:=stLine_BA02PL,
stStation:=stLine_BA02PL.stStation_BA02PL01,
stMachine:=stLine_BA02PL.stStation_BA02PL01.stMachine_1,
stSlaveParms:=GVL.st_Filler_A_Parameters,bNextMachineWork := TRUE);
END_ACTION

ACTION ACT_2_Cork:
GVL.st_Cork_Parameters.bPartsCount:= TRUE;
GVL.st_Cork_Parameters.iErrorOffset := 1100;
GVL.st_Cork_Parameters.iPort:= 500;
GVL.st_Cork_Parameters.iUnitId := 1;
GVL.st_Cork_Parameters.sIpAdress := '192.168.13.181';
GVL.st_Cork_Parameters.iRegisterReadStartAdress:=9000;
GVL.st_Cork_Parameters.iRegisterWriteStartAdress:=9020;
GVL.st_Cork_Parameters.iRegisterReadAmount := 20;
GVL.st_Cork_Parameters.iRegisterWriteAmount := 20;
GVL.st_Cork_Parameters.sMachineIdenfier := 'BA02PL01_M2';


fb_Cork_Machine(
stLine:=stLine_BA02PL,
stStation:=stLine_BA02PL.stStation_BA02PL01,
stMachine:=stLine_BA02PL.stStation_BA02PL01.stMachine_2,
stSlaveParms:=GVL.st_Cork_Parameters,bNextMachineWork := TRUE);
END_ACTION

ACTION ACT_3_SonicTech:
fb_1_SonicTech_SonictechUSW(
	stLine:=stLine_BA02PL,
	stStation:=stLine_BA02PL.stStation_BA02PL02,
	stMachine:=stLine_BA02PL.stStation_BA02PL02.stMachine_1,
	stDigitalInOut:= GVL_IO.st_1_SonicTech_WeldingMachine_IO, 
	I_Fix := ,
	fbCoreModbus := fbModbusCoreS02_S04,
	stMachineSettings:= GVL.st_1_SonicTech_USWelderSettings);
END_ACTION

ACTION ACT_4_Filler_B:
GVL.st_Filler_B_Parameters.bPartsCount:= TRUE;
GVL.st_Filler_B_Parameters.iErrorOffset := 1000;
GVL.st_Filler_B_Parameters.iPort:= 500;
GVL.st_Filler_B_Parameters.iUnitId := 1;
GVL.st_Filler_B_Parameters.sIpAdress := '192.168.13.182';
GVL.st_Filler_B_Parameters.iRegisterReadStartAdress:=9000;
GVL.st_Filler_B_Parameters.iRegisterWriteStartAdress:=9020;
GVL.st_Filler_B_Parameters.iRegisterReadAmount := 20;
GVL.st_Filler_B_Parameters.iRegisterWriteAmount := 20;
GVL.st_Filler_B_Parameters.sMachineIdenfier := 'BA02PL03';

fb_Filler_B_Machine(
stLine:=stLine_BA02PL,
stStation:=stLine_BA02PL.stStation_BA02PL03,
stMachine:=stLine_BA02PL.stStation_BA02PL03.stMachine_1,
stSlaveParms:=GVL.st_Filler_B_Parameters,bNextMachineWork := TRUE);
END_ACTION

ACTION ACT_5_SonicTech:
fb_2_SonicTech_SonictechUSW(
	stLine:=stLine_BA02PL,
	stStation:=stLine_BA02PL.stStation_BA02PL04,
	stMachine:=stLine_BA02PL.stStation_BA02PL04.stMachine_1,
	stDigitalInOut:= GVL_IO.st_2_SonicTech_WeldingMachine_IO, 
	I_Fix := ,
	fbCoreModbus := fbModbusCoreS02_S04,
	stMachineSettings:= GVL.st_2_SonicTech_USWelderSettings);
END_ACTION

ACTION ACT_6_UnderPressure_Tester:

fb_UnderPressure_Tester_Machine(
	stLine:=stLine_BA02PL,
	stStation:=stLine_BA02PL.stStation_BA02PL05,
	stMachine:=stLine_BA02PL.stStation_BA02PL05.stMachine_1);

fbTransporterUnderpressure(	stInOuts:=GVL_IO.stTransporterInOuts,
							fbChamber:=fb_UnderPressure_Tester_Machine);
END_ACTION

ACTION ACT_7_Sticker:
GVL.st_Sticker_Parameters.bPartsCount:= FALSE;
GVL.st_Sticker_Parameters.iErrorOffset := 1200;
GVL.st_Sticker_Parameters.iPort:= 500;
GVL.st_Sticker_Parameters.iUnitId := 1;
GVL.st_Sticker_Parameters.sIpAdress := '192.168.13.183';
GVL.st_Sticker_Parameters.iRegisterReadStartAdress:=9000;
GVL.st_Sticker_Parameters.iRegisterWriteStartAdress:=9020;
GVL.st_Sticker_Parameters.iRegisterReadAmount := 20;
GVL.st_Sticker_Parameters.iRegisterWriteAmount := 20;
GVL.st_Sticker_Parameters.sMachineIdenfier := 'BA02PL06_M1';

fb_Sticker_Machine(
stLine:=stLine_BA02PL,
stStation:=stLine_BA02PL.stStation_BA02PL06,
stMachine:=stLine_BA02PL.stStation_BA02PL06.stMachine_1,
stSlaveParms:=GVL.st_Sticker_Parameters,bNextMachineWork :=fb_Laser_Machine.stPimCommunicationData.bWorkInProgress);
END_ACTION

ACTION ACT_8_Laser:
GVL.st_Laser_Parameters.bPartsCount:= TRUE;
GVL.st_Laser_Parameters.iErrorOffset := 1300;
GVL.st_Laser_Parameters.iPort:= 500;
GVL.st_Laser_Parameters.iUnitId := 1;
GVL.st_Laser_Parameters.sIpAdress := '192.168.13.184';
GVL.st_Laser_Parameters.iRegisterReadStartAdress:=9000;
GVL.st_Laser_Parameters.iRegisterWriteStartAdress:=9020;
GVL.st_Laser_Parameters.iRegisterReadAmount := 20;
GVL.st_Laser_Parameters.iRegisterWriteAmount := 20;
GVL.st_Laser_Parameters.sMachineIdenfier := 'BA02PL06_M2';

fb_Laser_Machine(
stLine:=stLine_BA02PL,
stStation:=stLine_BA02PL.stStation_BA02PL06,
stMachine:=stLine_BA02PL.stStation_BA02PL06.stMachine_2,
stSlaveParms:=GVL.st_Laser_Parameters,bNextMachineWork := MAIN.fbWeighingTunel.fbTableControl.fbPIM.prWorkPermission,fbTCP_Send:=fb_Laser_TCP);

fb_Laser_TCP_Manual.bExecute;
fb_Laser_TCP_Manual(sRemoteHostIP:='192.168.1.234',nRemotePort:=45678,sDataToSend:='OpenDoc,MERCEDES.bpd',sSuffix:=';;');
fb_Laser_TCP();
END_ACTION

ACTION ACT_9_WeighingTunel:


fbSmartCamera.prManualMode:=fbWeighingTunel.fbWeighingStation.bManualModeActive;

fbSmartCamera(stParams:=stSmartCameraParams);
fbWeighingTunel(	
stLine:=stLine_BA02PL,
stStation:=stLine_BA02PL.stStation_BA02PL07,
stMachine:=stLine_BA02PL.stStation_BA02PL07.stMachine_1,
fbVision:=fbSmartCamera);
END_ACTION

ACTION ACT_HP1:
fbHotPlate_G1_M1(
	stLine:=stLine_BH0GPL,
	stStation:=stLine_BH0GPL.stStation_BH0GPL01,
	stMachine:=stLine_BH0GPL.stStation_BH0GPL01.stMachine_1,
	bMarkingAsembled := FALSE, 
	bELM := TRUE);

fbHotPlate_G1_M2(
	stLine:=stLine_BH0GPL,
	stStation:=stLine_BH0GPL.stStation_BH0GPL01,
	stMachine:=stLine_BH0GPL.stStation_BH0GPL01.stMachine_2,
	bMarkingAsembled := FALSE, 
	bELM := TRUE);

fbHotPlate_G1_M3(
	stLine:=stLine_BH0GPL,
	stStation:=stLine_BH0GPL.stStation_BH0GPL01,
	stMachine:=stLine_BH0GPL.stStation_BH0GPL01.stMachine_3,
	bMarkingAsembled := TRUE, 
	bELM := TRUE);
END_ACTION

ACTION ACT_HP2:
fbHotPlate_G2_M1(
	stLine:=stLine_BH0HPL,
	stStation:=stLine_BH0HPL.stStation_BH0HPL01,
	stMachine:=stLine_BH0HPL.stStation_BH0HPL01.stMachine_1,
	bMarkingAsembled := FALSE, 
	bELM := TRUE);

fbHotPlate_G2_M2(
	stLine:=stLine_BH0HPL,
	stStation:=stLine_BH0HPL.stStation_BH0HPL01,
	stMachine:=stLine_BH0HPL.stStation_BH0HPL01.stMachine_2,
	bMarkingAsembled := FALSE, 
	bELM := TRUE);

fbHotPlate_G2_M3(
	stLine:=stLine_BH0HPL,
	stStation:=stLine_BH0HPL.stStation_BH0HPL01,
	stMachine:=stLine_BH0HPL.stStation_BH0HPL01.stMachine_3,
	bMarkingAsembled := TRUE, 
	bELM := TRUE);
END_ACTION

ACTION ACT_HP3:
fbHotPlate_G3_M1(
	stLine:=stLine_BH0IPL,
	stStation:=stLine_BH0IPL.stStation_BH0IPL01,
	stMachine:=stLine_BH0IPL.stStation_BH0IPL01.stMachine_1,
	bMarkingAsembled := FALSE, 
	bELM := TRUE);

fbHotPlate_G3_M2(
	stLine:=stLine_BH0IPL,
	stStation:=stLine_BH0IPL.stStation_BH0IPL01,
	stMachine:=stLine_BH0IPL.stStation_BH0IPL01.stMachine_2,
	bMarkingAsembled := FALSE, 
	bELM := TRUE);

fbHotPlate_G3_M3(
	stLine:=stLine_BH0IPL,
	stStation:=stLine_BH0IPL.stStation_BH0IPL01,
	stMachine:=stLine_BH0IPL.stStation_BH0IPL01.stMachine_3,
	bMarkingAsembled := TRUE, 
	bELM := TRUE);
END_ACTION

ACTION ACT_HP4:
fbHotPlate_G4_M1(
	stLine:=stLine_BH0JPL,
	stStation:=stLine_BH0JPL.stStation_BH0JPL01,
	stMachine:=stLine_BH0JPL.stStation_BH0JPL01.stMachine_1,
	bMarkingAsembled := FALSE, 
	bELM := TRUE);

fbHotPlate_G4_M2(
	stLine:=stLine_BH0JPL,
	stStation:=stLine_BH0JPL.stStation_BH0JPL01,
	stMachine:=stLine_BH0JPL.stStation_BH0JPL01.stMachine_2,
	bMarkingAsembled := FALSE, 
	bELM := TRUE);

fbHotPlate_G4_M3(
	stLine:=stLine_BH0JPL,
	stStation:=stLine_BH0JPL.stStation_BH0JPL01,
	stMachine:=stLine_BH0JPL.stStation_BH0JPL01.stMachine_3,
	bMarkingAsembled := TRUE, 
	bELM := TRUE);
END_ACTION

ACTION ACT_HP5:
fbHotPlate_G5_M1(
	stLine:=stLine_BH0KPL,
	stStation:=stLine_BH0KPL.stStation_BH0KPL01,
	stMachine:=stLine_BH0KPL.stStation_BH0KPL01.stMachine_1,
	bMarkingAsembled := FALSE, 
	bELM := TRUE);

fbHotPlate_G5_M2(
	stLine:=stLine_BH0KPL,
	stStation:=stLine_BH0KPL.stStation_BH0KPL01,
	stMachine:=stLine_BH0KPL.stStation_BH0KPL01.stMachine_2,
	bMarkingAsembled := FALSE, 
	bELM := TRUE);

fbHotPlate_G5_M3(
	stLine:=stLine_BH0KPL,
	stStation:=stLine_BH0KPL.stStation_BH0KPL01,
	stMachine:=stLine_BH0KPL.stStation_BH0KPL01.stMachine_3,
	bMarkingAsembled := TRUE, 
	bELM := TRUE);
END_ACTION

ACTION ACT_HP6:
fbHotPlate_G6_M1(
	stLine:=stLine_BH0LPL,
	stStation:=stLine_BH0LPL.stStation_BH0LPL01,
	stMachine:=stLine_BH0LPL.stStation_BH0LPL01.stMachine_1,
	bMarkingAsembled := FALSE, 
	bELM := TRUE);

fbHotPlate_G6_M2(
	stLine:=stLine_BH0LPL,
	stStation:=stLine_BH0LPL.stStation_BH0LPL01,
	stMachine:=stLine_BH0LPL.stStation_BH0LPL01.stMachine_2,
	bMarkingAsembled := FALSE, 
	bELM := TRUE);

fbHotPlate_G6_M3(
	stLine:=stLine_BH0LPL,
	stStation:=stLine_BH0LPL.stStation_BH0LPL01,
	stMachine:=stLine_BH0LPL.stStation_BH0LPL01.stMachine_3,
	bMarkingAsembled := TRUE, 
	bELM := TRUE);
END_ACTION

ACTION ACT_HP7:
fbHotPlate_G7_M1(
	stLine:=stLine_BH0MPL,
	stStation:=stLine_BH0MPL.stStation_BH0MPL01,
	stMachine:=stLine_BH0MPL.stStation_BH0MPL01.stMachine_1,
	bMarkingAsembled := FALSE, 
	bELM := TRUE);

fbHotPlate_G7_M2(
	stLine:=stLine_BH0MPL,
	stStation:=stLine_BH0MPL.stStation_BH0MPL01,
	stMachine:=stLine_BH0MPL.stStation_BH0MPL01.stMachine_2,
	bMarkingAsembled := FALSE, 
	bELM := TRUE);

fbHotPlate_G7_M3(
	stLine:=stLine_BH0MPL,
	stStation:=stLine_BH0MPL.stStation_BH0MPL01,
	stMachine:=stLine_BH0MPL.stStation_BH0MPL01.stMachine_3,
	bMarkingAsembled := TRUE, 
	bELM := TRUE);
END_ACTION

ACTION ACT_S01:
// Prasa ze zgrzewarki Sonictech
fbS01_BearingPress(
	stLine:=stLine_BS02PL,
	stStation:=stLine_BS02PL.stStation_BS02PL01,
	stMachine:=stLine_BS02PL.stStation_BS02PL01.stMachine_1,
	stDigInOuts := GVL_IO.stS01_1_BearingPress_IO,
	I_Fix := fbS01_KeyencePNVisSens,
	stTestParams:= GVL.stS01_TestParams,
	stMachineSettings:= GVL.stS01_PressSettings);
	
fbS01_KeyencePNVisSens(I_Sonic:=fbS01_BearingPress,
	stParams := );
	
IF bTrigger THEN
	GVL_IO.bS01_Trigger := TRUE;
	bTrigger := FALSE;
ELSE	
	GVL_IO.bS01_Trigger := FALSE;	
END_IF
END_ACTION

ACTION ACT_S02:

// Prasa ze zgrzewarki Sonictech
fbS02_BearingPress(
	stLine:=stLine_BB02PL,
	stStation:=stLine_BB02PL.stStation_BB02PL01,
	stMachine:=stLine_BB02PL.stStation_BB02PL01.stMachine_1,
	stDigInOuts := GVL_IO.stS02_1_BearingPress_IO,
	I_Fix := 0,
	stTestParams:= GVL.stS02_TestParams,
	stMachineSettings:= GVL.stS02_PressSettings);
END_ACTION

ACTION ACT_S03:
// Prasa ze zgrzewarki Sonictech
fbS03_BearingPress(
	stLine:=stLine_BO02PL,
	stStation:=stLine_BO02PL.stStation_BO02PL01,
	stMachine:=stLine_BO02PL.stStation_BO02PL01.stMachine_1,
	stDigInOuts := GVL_IO.stS03_1_BearingPress_IO,
	I_Fix := fbS03_CapFixture,
	stTestParams:= GVL.stS03_TestParams,
	stMachineSettings:= GVL.stS03_PressSettings);
	
fbS03_CapFixture(I_Sonic:=fbS03_BearingPress,stInOuts:=GVL_IO.stS03_CapFixture_IO);
END_ACTION

ACTION ACT_S04:
// Prasa ze zgrzewarki Sonictech
fbS04_BearingPress(
	stLine:=stLine_BO02PL,
	stStation:=stLine_BO02PL.stStation_BO02PL02,
	stMachine:=stLine_BO02PL.stStation_BO02PL02.stMachine_1,
	stDigInOuts := GVL_IO.stS04_1_BearingPress_IO,
	I_Fix := 0,
	stTestParams:= GVL.stS04_TestParams,
	stMachineSettings:= GVL.stS04_PressSettings);
END_ACTION

ACTION ACT_SafetyBackupRestore:
//fbEL6910Backup(
END_ACTION

END_PROGRAM

// ---- POUs/SafetyBackupRestore.TcPOU
PROGRAM SafetyBackupRestore
VAR
	wSafetyProjectCRC AT %I*: WORD;
	udiSafetyPLCSerialNb AT %I*: UDINT;
	fbEL6910Backup: FB_SAVELOGICPROGRAM;
	fbEL6910Restore: FB_RESTORELOGICPROGRAM;
	bStartBackup: BOOL;
	abEL6910AmsNetID AT %I*: ARRAY [0..5] OF BYTE;
	wEL6910port AT %I*: WORD;
	abInternalBuffer: ARRAY[0..16#FFFF] OF BYTE;
	sFileString: T_MaxString := 'c:\temp\safety\complibTest_EL6910.bin';
	LocalAmsNetID: T_AmsNetID := '172.55.76.53.1.1';
	bSaveDone: BOOL;
	sSaveResult: STRING(200);
	bSaveErr: BOOL;
	bStartRestore: BOOL;
	abInternalbuffer2: ARRAY[0..16#FFFF] OF BYTE;
	bRestoreDone: BOOL;
	sRestoreResult: STRING(200);
	bRestoreErr: BOOL;
END_VAR

END_PROGRAM

// ---- POUs/Program_PIM_Lines/B02PL_LineBackground.TcPOU
PROGRAM B02PL_LineBackground
VAR
END_VAR

BA02PL_LineBackground();
BB02PL_LineBackground();
BS02PL_LineBackground();
BO02PL_LineBackground();
BH0GPL_LineBackground();
BH0HPL_LineBackground();
BH0IPL_LineBackground();
BH0JPL_LineBackground();
BH0KPL_LineBackground();
BH0LPL_LineBackground();
BH0MPL_LineBackground();

END_PROGRAM

// ---- POUs/Program_PIM_Lines/Filling/BA02PL_LineBackground.TcPOU
PROGRAM BA02PL_LineBackground
VAR
END_VAR

MAIN.stLine_BA02PL.fbLine(stLine:=MAIN.stLine_BA02PL,bMainLine:=TRUE);
MAIN.stLine_BA02PL.stStation_BA02PL01.fbStation(
				stLine:=MAIN.stLine_BA02PL,
				stStation:=MAIN.stLine_BA02PL.stStation_BA02PL01);
MAIN.stLine_BA02PL.stStation_BA02PL02.fbStation(
				stLine:=MAIN.stLine_BA02PL,
				stStation:=MAIN.stLine_BA02PL.stStation_BA02PL02);
MAIN.stLine_BA02PL.stStation_BA02PL03.fbStation(
				stLine:=MAIN.stLine_BA02PL,
				stStation:=MAIN.stLine_BA02PL.stStation_BA02PL03);
MAIN.stLine_BA02PL.stStation_BA02PL04.fbStation(
				stLine:=MAIN.stLine_BA02PL,
				stStation:=MAIN.stLine_BA02PL.stStation_BA02PL04);
MAIN.stLine_BA02PL.stStation_BA02PL05.fbStation( 
				stLine:=MAIN.stLine_BA02PL,
				stStation:=MAIN.stLine_BA02PL.stStation_BA02PL05);
MAIN.stLine_BA02PL.stStation_BA02PL06.fbStation(
				stLine:=MAIN.stLine_BA02PL,
				stStation:=MAIN.stLine_BA02PL.stStation_BA02PL06);
MAIN.stLine_BA02PL.stStation_BA02PL07.fbStation(
				stLine:=MAIN.stLine_BA02PL,
				stStation:=MAIN.stLine_BA02PL.stStation_BA02PL07);

END_PROGRAM

// ---- POUs/Program_PIM_Lines/PreAssembly/BB02PL_LineBackground.TcPOU
PROGRAM BB02PL_LineBackground
VAR
END_VAR

MAIN.stLine_BB02PL.fbLine(stLine:=MAIN.stLine_BB02PL);
MAIN.stLine_BB02PL.stStation_BB02PL01.fbStation(
				stLine:=MAIN.stLine_BB02PL,
				stStation:=MAIN.stLine_BB02PL.stStation_BB02PL01);

END_PROGRAM

// ---- POUs/Program_PIM_Lines/PreAssembly/BS02PL_LineBackground.TcPOU
PROGRAM BS02PL_LineBackground
VAR
END_VAR

MAIN.stLine_BS02PL.fbLine(stLine:=MAIN.stLine_BS02PL);
MAIN.stLine_BS02PL.stStation_BS02PL01.fbStation(
				stLine:=MAIN.stLine_BS02PL,
				stStation:=MAIN.stLine_BS02PL.stStation_BS02PL01);

END_PROGRAM

// ---- POUs/Program_PIM_Lines/PreAssembly/BO02PL_LineBackground.TcPOU
PROGRAM BO02PL_LineBackground
VAR
END_VAR

MAIN.stLine_BO02PL.fbLine(stLine:=MAIN.stLine_BO02PL);
MAIN.stLine_BO02PL.stStation_BO02PL01.fbStation(
				stLine:=MAIN.stLine_BO02PL,
				stStation:=MAIN.stLine_BO02PL.stStation_BO02PL01);
MAIN.stLine_BO02PL.stStation_BO02PL02.fbStation(
				stLine:=MAIN.stLine_BO02PL,
				stStation:=MAIN.stLine_BO02PL.stStation_BO02PL02);

END_PROGRAM

// ---- POUs/Program_PIM_Lines/HP/BH0GPL_LineBackground.TcPOU
PROGRAM BH0GPL_LineBackground
VAR
END_VAR

MAIN.stLine_BH0GPL.fbLine(stLine:=MAIN.stLine_BH0GPL);
MAIN.stLine_BH0GPL.stStation_BH0GPL01.fbStation(
				stLine:=MAIN.stLine_BH0GPL,
				stStation:=MAIN.stLine_BH0GPL.stStation_BH0GPL01);

END_PROGRAM

// ---- POUs/Program_PIM_Lines/HP/BH0HPL_LineBackground.TcPOU
PROGRAM BH0HPL_LineBackground
VAR
END_VAR

MAIN.stLine_BH0GPL.fbLine(stLine:=MAIN.stLine_BH0GPL);
MAIN.stLine_BH0GPL.stStation_BH0GPL01.fbStation(
				stLine:=MAIN.stLine_BH0GPL,
				stStation:=MAIN.stLine_BH0GPL.stStation_BH0GPL01);

END_PROGRAM

// ---- POUs/Program_PIM_Lines/HP/BH0IPL_LineBackground.TcPOU
PROGRAM BH0IPL_LineBackground
VAR
END_VAR

